DATA_BLOCK "INOUT"	// DB 80
VERSION : 0.1
  STRUCT
   I_TRO : STRUCT
    Fuse_115V_OK : BOOL ;	//115V AC OK
    Fuse_24V_OK : BOOL ;	//fuse 24V DC OK
    Overtemp_Cabinet : BOOL ;	//high temperature cabinet
    PowerBrakes_OK : BOOL ;	//Power supply brakes OK
    Power_Lift_OK : BOOL ;	//Power supply lift OK
    Power_Drum_OK : BOOL ;	//Power supply cable drum OK
    TRO_Power_Cabinet_Fan : BOOL ;	//Power supply cabinet fan OK
    TRO_Cabinet_Fan_ON : BOOL ;	//cabinet fan running
    BTN_Reset : BOOL ;	//Reset button (top cabinet)
    BTN_Preset : BOOL ;	//Preset button (3s)
    Preset_Bit_0 : BOOL ;	//Preset selection switch bit 0
    Preset_Bit_1 : BOOL ;	//Preset selection switch bit 1
    Preset_Bit_2 : BOOL ;	//Preset selection switch bit 2
    Preset_Bit_3 : BOOL ;	//Preset selection switch bit 3
    E76_6 : BOOL ;	//spare
    E76_7 : BOOL ;	//spare
    check_cableDrum_NO : BOOL ;	//check cable drum NO
    check_cableDrum_NC : BOOL ;	//check cable drum NC
    E77_2 : BOOL ;	//spar
    E77_3 : BOOL ;	//spar
    Buffer_left_Free : BOOL ;	//Buffer left occupied
    Buffer_right_Free : BOOL ;	//Buffer right occupied
    LIF_Limit_TOP : BOOL ;	//Lift limit switch top (minus)
    LIF_Limit_BOTTOM : BOOL ;	//Lift limit switch bottom (plus)
    LIF_Pos_TOP_NO : BOOL ;	//Lift limit prox. top NO
    LIF_Pos_TOP_NC : BOOL ;	//Lift limit prox. top NC
    Limit_plus : BOOL ;	//Tolley limit switch plus
    Limit_minus : BOOL ;	//Tolley limit switch minus
    FS_plus_NO : BOOL ;	//Tolley prox. switch forced slow plus NO
    FS_plus_NC : BOOL ;	//Tolley prox. switch forced slow plus NC
    FS_minus_NO : BOOL ;	//Tolley prox. switch forced slow minus NO
    FS_minus_NC : BOOL ;	//Tolley prox. switch forced slow minus NC
    SSI_Barcode_noPos : BOOL ;	//Datamatrix SSI error: no position
    SSI_Barcode_dirty : BOOL ;	//Datamatrix SSI error: dirty
    Profinet_Barcode_noPos : BOOL ;	//Datamatrix Profinet error: no position
    Profinet_Barcode_dirty : BOOL ;	//Datamatrix Profinet error: dirty
    FallProtection_Pl_1 : BOOL ;	//Trooley plus fall protection ch1
    FallProtection_Pl_2 : BOOL ;	//Trooley plus fall protection ch12
    FallProtection_Mi_1 : BOOL ;	//Trooley minus fall protection ch1
    FallProtection_Mi_2 : BOOL ;	//Trooley minus fall protection ch2
    Plus : BOOL ;	//Trolley drive plus
    Minus : BOOL ;	//Trolley drive minus
    Lift_up : BOOL ;	//Lift drive up
    Lift_down : BOOL ;	//Lift drive down
    TEL_Plus : BOOL ;	//Tellescope drive plus
    TEL_Minus : BOOL ;	//Tellescope drive minus
    E80_6 : BOOL ;	//spare
    E80_7 : BOOL ;	//spare
    spare : ARRAY  [1 .. 4 ] OF WORD ;
   END_STRUCT ;
   O_TRO : STRUCT
    A75_0 : BOOL ;	//spare
    Reset_24V : BOOL ;	//reset 24V fuses
    E75_02 : BOOL ;	//spare
    LP_Reset : BOOL ;	//lamp reset
    E75_4 : BOOL ;	//spare
    CableDrum : BOOL ;	//start cable drum
    EStop_Reset : BOOL ;	//ESTOP reset
    LP_Preset : BOOL ;	//lamp preset
    Horn : BOOL ;	//startup warning
    LP_State_0 : BOOL ;	//lamp state 0
    LP_State_1 : BOOL ;	//lamp state 1
    LP_State_2 : BOOL ;	//lamp state 2
    E76_4 : BOOL ;	//spare
    SEW_Reset : BOOL ;	//reset movi PLC
    EmergencyMode : BOOL ;	//Emergency Mode
    LIF_StartFan : BOOL ;	//startup Lift Fan
    EmergencyMode_Fwd : BOOL ;	//Emergency mode forward
    EmergencyMode_Bwd : BOOL ;	//Emergency mode backward
    A77_2 : BOOL ;	//startup Lift Fan
    A77_3 : BOOL ;	//Emergency mode forward
    A77_4 : BOOL ;	//Emergency mode backward
    A77_5 : BOOL ;	//spare
    A77_6 : BOOL ;	//spare
    A77_7 : BOOL ;	//spare
    spar_1 : BOOL ;	//spare
    spare_2 : BOOL ;	//spare
    spare_3 : BOOL ;	//spare
    spare : ARRAY  [1 .. 2 ] OF WORD ;
   END_STRUCT ;
   I_LIF : STRUCT
    E85_0 : BOOL ;	//spare
    E85_1 : BOOL ;	//spare
    E85_2 : BOOL ;	//spare
    E85_3 : BOOL ;	//spare
    error_NO : BOOL ;	//Drive telescopes error NO
    error_NC : BOOL ;	//Drive telescopes error NC
    E85_6 : BOOL ;	//spare
    E85_7 : BOOL ;	//spare
    Overload_L_NO : BOOL ;	//Overload-Monitoring left NO
    Overload_R_NO : BOOL ;	//Overload-Monitoring rigth NO
    SlapRope_L_NO : BOOL ;	//Slap-Rope-Monitoring left NO
    SlapRope_R_NO : BOOL ;	//Slap-Rope-Monitoring right NO
    E86_4 : BOOL ;	//spare
    E86_5 : BOOL ;	//spare
    TEL_Front_FirstHookOcc : BOOL ;	//hook front left occupied (1)
    TEL_Front_LastHookOcc : BOOL ;	//hook rear left occupied (2)
    TEL_Rear_FirstHookOcc : BOOL ;	//hook front right occupied (11)
    TEL_Rear_LastHookOcc : BOOL ;	//hook rear right occupied (12)
    E87_2 : BOOL ;	//spare
    E87_3 : BOOL ;	//spare
    TEL_inMidle_L : BOOL ;	//telescope left in middle position
    TEL_inMidle_R : BOOL ;	//telescope right in middle position
    E87_6 : BOOL ;	//spare
    TEL_Left_Occ_NO : BOOL ;	//telescope left occupied NO
    E88_0 : BOOL ;	//spare
    TEL_Right_Occ_NO : BOOL ;	//telescope right occupied NO
    TEL_Limit_front_NO : BOOL ;	//telescopes limit switch front NO
    TEL_Limit_front_NC : BOOL ;	//telescopes limit switch front NC
    TEL_Limit_back_NO : BOOL ;	//telescopes limit switch back NO
    TEL_Limit_back_NC : BOOL ;	//telescopes limit switch back NC
    E88_6 : BOOL ;	//spare
    E88_7 : BOOL ;	//spare
    E89_0 : BOOL ;	//spare
    E89_1 : BOOL ;	//spare
    E89_2 : BOOL ;	//spare
    E89_3 : BOOL ;	//spare
    E89_4 : BOOL ;	//spare
    E89_5 : BOOL ;	//spare
    E89_6 : BOOL ;	//spare
    E89_7 : BOOL ;	//spare
    TEL_Encoder : DINT ;	//Teleskope Encoder
   END_STRUCT ;
   O_LIF : STRUCT
    TEL_Mode1 : BOOL ;	//telescope mode_1
    TEL_Mode2 : BOOL ;	//telescope mode_2
    TEL_Start : BOOL ;	//start telescope
    TEL_Reset : BOOL ;	//reset telescope
    TEL_BCD_Bit_1 : BOOL ;	//telescope BCD Bit_1
    TEL_BCD_Bit_2 : BOOL ;	//telescope BCD Bit_2
    TEL_BCD_Bit_3 : BOOL ;	//telescope BCD Bit_3
    TEL_BCD_Bit_4 : BOOL ;	//telescope BCD Bit_4
    TEL_Light_Front_Left : BOOL ;	//lightning telescopes front left on
    TEL_Light_Front_Rigth : BOOL ;	//lightning telescopes front rigth on
    TEL_Light_Rear_Left : BOOL ;	//lightning telescopes rear Left on
    TEL_Light_Rear_Rigth : BOOL ;	//lightning telescopes rigth on
    TEL_Preset_Telescope : BOOL ;	//Preset Encoder Telescope
    A86_5 : BOOL ;	//spare
    A86_6 : BOOL ;	//spare
    A86_7 : BOOL ;	//spare
    A87_0 : BOOL ;	//spare
    A87_1 : BOOL ;	//spare
    A87_2 : BOOL ;	//spare
    A87_3 : BOOL ;	//spare
    A87_4 : BOOL ;	//spare
    A87_5 : BOOL ;	//spare
    A87_6 : BOOL ;	//spare
    A87_7 : BOOL ;	//spare
   END_STRUCT ;
  END_STRUCT ;	
BEGIN
   I_TRO.Fuse_24V_OK := TRUE;
   I_TRO.PowerBrakes_OK := TRUE;
   I_TRO.Power_Lift_OK := TRUE;
   I_TRO.Power_Drum_OK := TRUE;
   I_TRO.TRO_Power_Cabinet_Fan := TRUE;
   I_TRO.TRO_Cabinet_Fan_ON := TRUE;
   I_TRO.check_cableDrum_NO := TRUE;
   I_TRO.LIF_Pos_TOP_NO := TRUE;
   O_TRO.LP_State_0 := TRUE;
   I_LIF.error_NO := TRUE;
   I_LIF.error_NC := TRUE;
   I_LIF.TEL_Front_FirstHookOcc := TRUE;
   I_LIF.TEL_Front_LastHookOcc := TRUE;
   I_LIF.TEL_inMidle_L := TRUE;
   I_LIF.TEL_inMidle_R := TRUE;
   I_LIF.TEL_Left_Occ_NO := TRUE;
   I_LIF.TEL_Right_Occ_NO := TRUE;
   I_LIF.TEL_Limit_front_NC := TRUE;
   I_LIF.TEL_Limit_back_NC := TRUE;
   O_LIF.TEL_Mode2 := TRUE;
END_DATA_BLOCK

DATA_BLOCK "DB_ActualHookdata"	// DB 92
VERSION : 0.1
  STRUCT
   Front : STRUCT
    Hook : ARRAY  [1 .. 10 ] OF UDT 102;
   END_STRUCT ;
   Rear : STRUCT
    Hook : ARRAY  [1 .. 10 ] OF UDT 102;
   END_STRUCT ;
   ActualDB_No : INT ;
  END_STRUCT ;	
BEGIN
   Front.Hook[1].HookOver := L#6716;
   Front.Hook[1].HookUnderOffset := L#115;
   Front.Hook[1].TelPos_1.TelPos := L#3;
   Front.Hook[2].HookOver := L#5745;
   Front.Hook[2].HookUnderOffset := L#115;
   Front.Hook[2].TelPos_1.TelPos := L#3;
   Front.Hook[3].HookOver := L#4775;
   Front.Hook[3].HookUnderOffset := L#115;
   Front.Hook[3].TelPos_1.TelPos := L#3;
   Front.Hook[4].HookOver := L#3805;
   Front.Hook[4].HookUnderOffset := L#115;
   Front.Hook[4].TelPos_1.TelPos := L#3;
   Front.Hook[5].HookOver := L#2835;
   Front.Hook[5].HookUnderOffset := L#115;
   Front.Hook[5].TelPos_1.TelPos := L#3;
   Front.Hook[6].HookOver := L#1865;
   Front.Hook[6].HookUnderOffset := L#115;
   Front.Hook[6].TelPos_1.TelPos := L#3;
   Rear.Hook[1].HookOver := L#6716;
   Rear.Hook[1].HookUnderOffset := L#115;
   Rear.Hook[1].TelPos_1.TelPos := L#4;
   Rear.Hook[2].HookOver := L#5745;
   Rear.Hook[2].HookUnderOffset := L#115;
   Rear.Hook[2].TelPos_1.TelPos := L#4;
   Rear.Hook[3].HookOver := L#4775;
   Rear.Hook[3].HookUnderOffset := L#115;
   Rear.Hook[3].TelPos_1.TelPos := L#4;
   Rear.Hook[4].HookOver := L#3805;
   Rear.Hook[4].HookUnderOffset := L#115;
   Rear.Hook[4].TelPos_1.TelPos := L#4;
   Rear.Hook[5].HookOver := L#2835;
   Rear.Hook[5].HookUnderOffset := L#115;
   Rear.Hook[5].TelPos_1.TelPos := L#4;
   Rear.Hook[6].HookOver := L#1865;
   Rear.Hook[6].HookUnderOffset := L#115;
   Rear.Hook[6].TelPos_1.TelPos := L#4;
   ActualDB_No := 252;
END_DATA_BLOCK

DATA_BLOCK "Moves"	// DB 101
VERSION : 0.1
  STRUCT
   PC : UDT 7;
   Unit : ARRAY  [1 .. 50 ] OF UDT 7;
  END_STRUCT ;	
BEGIN
   PC.MsgCounter := 648;
   PC.Action := 4;
   PC.Value_01 := 5;
   PC.Value_02 := 8;
   PC.Value_03 := 100;
   PC.Value_04 := 100;
   Unit[1].Action := 4;
   Unit[1].Value_01 := 5;
   Unit[1].Value_02 := 8;
   Unit[1].Value_03 := 100;
   Unit[1].Value_04 := 100;
END_DATA_BLOCK

DATA_BLOCK "InstanzDB PNIODiag"	// DB 126
AUTHOR : ICom
FAMILY : DIAGNOSE
VERSION : 0.0
"PNIODiag"
BEGIN
END_DATA_BLOCK

DATA_BLOCK "InstanzDB STATDiag"	// DB 127
AUTHOR : ICom
FAMILY : DIAGNOSE
VERSION : 0.0
"STATDiag"
BEGIN
END_DATA_BLOCK

DATA_BLOCK "DB_Crane"	// DB 130
VERSION : 0.1
  STRUCT
   NoOfRows : INT  := 3;
   NoOfTowers : INT  := 13;
   NoOfPositions : INT  := 16;
   MoveCounts : DINT ;
   WorkingHours : DINT ;
   RemainigServiceHours : DINT ;
   CraneType : INT ;
   UnitNumber : INT ;
   Reserve9 : INT ;
   Reserve10 : INT ;
   Reserve11 : INT ;
   Reserve12 : INT ;
  END_STRUCT ;	
BEGIN
   NoOfRows := 3;
   NoOfTowers := 11;
   NoOfPositions := 16;
END_DATA_BLOCK

DATA_BLOCK "DB_Steps"	// DB 132
VERSION : 0.1
  STRUCT
   _DINT : STRUCT
    StepsStartet : DINT ;
    StepsFinished : DINT ;
    _02 : DINT ;
    _03 : DINT ;
    _04 : DINT ;
    _05 : DINT ;
    _06 : DINT ;
    _07 : DINT ;
    _08 : DINT ;
    _09 : DINT ;
    _10 : DINT ;
    _11 : DINT ;
    _12 : DINT ;
    _13 : DINT ;
    _14 : DINT ;
    _15 : DINT ;
    _16 : DINT ;
    _17 : DINT ;
    _18 : DINT ;
    _19 : DINT ;
    _20 : DINT ;
    _21 : DINT ;
    _22 : DINT ;
    _23 : DINT ;
    _24 : DINT ;
    _25 : DINT ;
    _26 : DINT ;
    _27 : DINT ;
    _28 : DINT ;
    _29 : DINT ;
    _30 : DINT ;
    _31 : DINT ;
    _32 : DINT ;
    _33 : DINT ;
    _34 : DINT ;
    _35 : DINT ;
    _36 : DINT ;
    _37 : DINT ;
    _38 : DINT ;
    _39 : DINT ;
    _40 : DINT ;
    _41 : DINT ;
    _42 : DINT ;
    _43 : DINT ;
    _44 : DINT ;
    _45 : DINT ;
    _46 : DINT ;
    _47 : DINT ;
    _48 : DINT ;
    _49 : DINT ;
    _50 : DINT ;
    _51 : DINT ;
    _52 : DINT ;
    _53 : DINT ;
    _54 : DINT ;
    _55 : DINT ;
    _56 : DINT ;
    _57 : DINT ;
    _58 : DINT ;
    _59 : DINT ;
    _60 : DINT ;
    _61 : DINT ;
    _62 : DINT ;
    _63 : DINT ;
    _64 : DINT ;
    _65 : DINT ;
    _66 : DINT ;
    _67 : DINT ;
    _68 : DINT ;
    _69 : DINT ;
    _70 : DINT ;
    _71 : DINT ;
    _72 : DINT ;
    _73 : DINT ;
    _74 : DINT ;
    _75 : DINT ;
    _76 : DINT ;
    _77 : DINT ;
    _78 : DINT ;
    _79 : DINT ;
    _80 : DINT ;
    _81 : DINT ;
    _82 : DINT ;
    _83 : DINT ;
    _84 : DINT ;
    _85 : DINT ;
    _86 : DINT ;
    _87 : DINT ;
    _88 : DINT ;
    _89 : DINT ;
    _90 : DINT ;
    _91 : DINT ;
    _92 : DINT ;
    _93 : DINT ;
    _94 : DINT ;
    _95 : DINT ;
    _96 : DINT ;
    _97 : DINT ;
    _98 : DINT ;
    _99 : DINT ;
    _100 : DINT ;
    _101 : DINT ;
    _102 : DINT ;
    _103 : DINT ;
    _104 : DINT ;
    _105 : DINT ;
    _106 : DINT ;
    _107 : DINT ;
    _108 : DINT ;
    _109 : DINT ;
    _110 : DINT ;
    _111 : DINT ;
    _112 : DINT ;
    _113 : DINT ;
    _114 : DINT ;
    _115 : DINT ;
    _116 : DINT ;
    _117 : DINT ;
    _118 : DINT ;
    _119 : DINT ;
    _120 : DINT ;
    _121 : DINT ;
    _122 : DINT ;
    _123 : DINT ;
    _124 : DINT ;
    _125 : DINT ;
    _126 : DINT ;
    _127 : DINT ;
    _128 : DINT ;
    _129 : DINT ;
    _130 : DINT ;
    _131 : DINT ;
    _132 : DINT ;
    _133 : DINT ;
    _134 : DINT ;
    _135 : DINT ;
    _136 : DINT ;
    _137 : DINT ;
    _138 : DINT ;
    _139 : DINT ;
    _140 : DINT ;
    _141 : DINT ;
    _142 : DINT ;
    _143 : DINT ;
    _144 : DINT ;
    _145 : DINT ;
    _146 : DINT ;
    _147 : DINT ;
    _148 : DINT ;
    _149 : DINT ;
    _150 : DINT ;
    _151 : DINT ;
    _152 : DINT ;
    _153 : DINT ;
    _154 : DINT ;
    _155 : DINT ;
    _156 : DINT ;
    _157 : DINT ;
    _158 : DINT ;
    _159 : DINT ;
   END_STRUCT ;
   _INT : STRUCT
    BASEPOS_Steps : INT ;
    EMPTY_Steps : INT ;
    GET_Steps : INT ;
    PUT_Steps : INT ;
    _04 : INT ;
    _05 : INT ;
    _06 : INT ;
    _07 : INT ;
    _08 : INT ;
    _09 : INT ;
    ChkHookOccCntGET : INT ;	//Check occupation sensors hook
    ChkHookOccCntPUT : INT ;
    _12 : INT ;
    _13 : INT ;
    _14 : INT ;
    _15 : INT ;
    _16 : INT ;
    _17 : INT ;
    _18 : INT ;
    _19 : INT ;
    _20 : INT ;
    _21 : INT ;
    _22 : INT ;
    _23 : INT ;
    _24 : INT ;
    _25 : INT ;
    _26 : INT ;
    _27 : INT ;
    _28 : INT ;
    _29 : INT ;
    _30 : INT ;
    _31 : INT ;
    _32 : INT ;
    _33 : INT ;
    _34 : INT ;
    _35 : INT ;
    _36 : INT ;
    _37 : INT ;
    _38 : INT ;
    _39 : INT ;
    _40 : INT ;
    _41 : INT ;
    _42 : INT ;
    _43 : INT ;
    _44 : INT ;
    _45 : INT ;
    _46 : INT ;
    _47 : INT ;
    _48 : INT ;
    _49 : INT ;
    _50 : INT ;
    _51 : INT ;
    _52 : INT ;
    _53 : INT ;
    _54 : INT ;
    _55 : INT ;
    _56 : INT ;
    _57 : INT ;
    _58 : INT ;
    _59 : INT ;
    _60 : INT ;
    _61 : INT ;
    _62 : INT ;
    _63 : INT ;
    _64 : INT ;
    _65 : INT ;
    _66 : INT ;
    _67 : INT ;
    _68 : INT ;
    _69 : INT ;
    _70 : INT ;
    _71 : INT ;
    _72 : INT ;
    _73 : INT ;
    _74 : INT ;
    _75 : INT ;
    _76 : INT ;
    _77 : INT ;
    _78 : INT ;
    _79 : INT ;
    _80 : INT ;
    _81 : INT ;
    _82 : INT ;
    _83 : INT ;
    _84 : INT ;
    _85 : INT ;
    _86 : INT ;
    _87 : INT ;
    _88 : INT ;
    _89 : INT ;
    _90 : INT ;
    _91 : INT ;
    _92 : INT ;
    _93 : INT ;
    _94 : INT ;
    _95 : INT ;
    _96 : INT ;
    _97 : INT ;
    _98 : INT ;
    _99 : INT ;
    _100 : INT ;
    _101 : INT ;
    _102 : INT ;
    _103 : INT ;
    _104 : INT ;
    _105 : INT ;
    _106 : INT ;
    _107 : INT ;
    _108 : INT ;
    _109 : INT ;
    _110 : INT ;
    _111 : INT ;
    _112 : INT ;
    _113 : INT ;
    _114 : INT ;
    _115 : INT ;
    _116 : INT ;
    _117 : INT ;
    _118 : INT ;
    _119 : INT ;
    _120 : INT ;
    _121 : INT ;
    _122 : INT ;
    _123 : INT ;
    _124 : INT ;
    _125 : INT ;
    _126 : INT ;
    _127 : INT ;
    _128 : INT ;
    _129 : INT ;
    _130 : INT ;
    _131 : INT ;
    _132 : INT ;
    _133 : INT ;
    _134 : INT ;
    _135 : INT ;
    _136 : INT ;
    _137 : INT ;
    _138 : INT ;
    _139 : INT ;
    _140 : INT ;
    _141 : INT ;
    _142 : INT ;
    _143 : INT ;
    _144 : INT ;
    _145 : INT ;
    _146 : INT ;
    _147 : INT ;
    _148 : INT ;
    _149 : INT ;
    _150 : INT ;
    _151 : INT ;
    _152 : INT ;
    _153 : INT ;
    _154 : INT ;
    _155 : INT ;
    _156 : INT ;
    _157 : INT ;
    _158 : INT ;
    _159 : INT ;
   END_STRUCT ;
   _BOOL : STRUCT
    Target_DataOK : BOOL ;
    _01 : BOOL ;
    _02 : BOOL ;
    _03 : BOOL ;
    _04 : BOOL ;
    _05 : BOOL ;
    _06 : BOOL ;
    _07 : BOOL ;
    BASEPOS_Req : BOOL ;
    EMPTY_Req : BOOL ;
    GET_Req : BOOL ;
    PUT_Req : BOOL ;
    BASEPOS_active : BOOL ;
    EMPTY_active : BOOL ;
    GET_active : BOOL ;
    PUT_active : BOOL ;
    STEPS_active : BOOL ;
    STEPS_start : BOOL ;
    GET_Finished : BOOL ;
    _19 : BOOL ;
    _20 : BOOL ;
    _21 : BOOL ;
    _22 : BOOL ;
    _23 : BOOL ;
    _24 : BOOL ;
    _25 : BOOL ;
    _26 : BOOL ;
    _27 : BOOL ;
    _28 : BOOL ;
    _29 : BOOL ;
    _30 : BOOL ;
    _31 : BOOL ;
    ChkHookOccGET : BOOL ;
    ChkHookOccGET_End : BOOL ;
    ChkHookOccGET_OK : BOOL ;
    ChkHookOccPUT : BOOL ;
    ChkHookOccPUT_End : BOOL ;
    ChkHookOccPUT_OK : BOOL ;
    ChkHookOcxGET_enable : BOOL ;
    ChkHookOcxPUT_enable : BOOL ;
    _40 : BOOL ;
    _41 : BOOL ;
    _42 : BOOL ;
    _43 : BOOL ;
    _44 : BOOL ;
    _45 : BOOL ;
    _46 : BOOL ;
    _47 : BOOL ;
    _48 : BOOL ;
    _49 : BOOL ;
    _50 : BOOL ;
    _51 : BOOL ;
    _52 : BOOL ;
    _53 : BOOL ;
    _54 : BOOL ;
    _55 : BOOL ;
    _56 : BOOL ;
    _57 : BOOL ;
    _58 : BOOL ;
    _59 : BOOL ;
    _60 : BOOL ;
    _61 : BOOL ;
    _62 : BOOL ;
    _63 : BOOL ;
    _64 : BOOL ;
    _65 : BOOL ;
    _66 : BOOL ;
    _67 : BOOL ;
    _68 : BOOL ;
    _69 : BOOL ;
    _70 : BOOL ;
    _71 : BOOL ;
    _72 : BOOL ;
    _73 : BOOL ;
    _74 : BOOL ;
    _75 : BOOL ;
    _76 : BOOL ;
    _77 : BOOL ;
    _78 : BOOL ;
    _79 : BOOL ;
    _80 : BOOL ;
    _81 : BOOL ;
    _82 : BOOL ;
    _83 : BOOL ;
    _84 : BOOL ;
    _85 : BOOL ;
    _86 : BOOL ;
    _87 : BOOL ;
    _88 : BOOL ;
    _89 : BOOL ;
    _90 : BOOL ;
    _91 : BOOL ;
    _92 : BOOL ;
    _93 : BOOL ;
    _94 : BOOL ;
    _95 : BOOL ;
    _96 : BOOL ;
    _97 : BOOL ;
    _98 : BOOL ;
    _99 : BOOL ;
    _100 : BOOL ;
    _101 : BOOL ;
    _102 : BOOL ;
    _103 : BOOL ;
    _104 : BOOL ;
    _105 : BOOL ;
    _106 : BOOL ;
    _107 : BOOL ;
    _108 : BOOL ;
    _109 : BOOL ;
    _110 : BOOL ;
    _111 : BOOL ;
    _112 : BOOL ;
    _113 : BOOL ;
    _114 : BOOL ;
    _115 : BOOL ;
    _116 : BOOL ;
    _117 : BOOL ;
    _118 : BOOL ;
    _119 : BOOL ;
    _120 : BOOL ;
    _121 : BOOL ;
    _122 : BOOL ;
    _123 : BOOL ;
    _124 : BOOL ;
    _125 : BOOL ;
    _126 : BOOL ;
    _127 : BOOL ;
    _128 : BOOL ;
    _129 : BOOL ;
    _130 : BOOL ;
    _131 : BOOL ;
    _132 : BOOL ;
    _133 : BOOL ;
    _134 : BOOL ;
    _135 : BOOL ;
    _136 : BOOL ;
    _137 : BOOL ;
    _138 : BOOL ;
    _139 : BOOL ;
    _140 : BOOL ;
    _141 : BOOL ;
    _142 : BOOL ;
    _143 : BOOL ;
    _144 : BOOL ;
    _145 : BOOL ;
    _146 : BOOL ;
    _147 : BOOL ;
    _148 : BOOL ;
    _149 : BOOL ;
    _150 : BOOL ;
    _151 : BOOL ;
    _152 : BOOL ;
    _153 : BOOL ;
    _154 : BOOL ;
    _155 : BOOL ;
    _156 : BOOL ;
    _157 : BOOL ;
    _158 : BOOL ;
    _159 : BOOL ;
   END_STRUCT ;
  END_STRUCT ;	
BEGIN
   _DINT.StepsStartet := L#46754;
   _DINT.StepsFinished := L#5503;
   _INT.GET_Steps := 50;
   _INT.ChkHookOccCntGET := 5;
   _INT.ChkHookOccCntPUT := 3;
   _BOOL.GET_active := TRUE;
   _BOOL.STEPS_active := TRUE;
   _BOOL.ChkHookOcxGET_enable := TRUE;
   _BOOL.ChkHookOcxPUT_enable := TRUE;
END_DATA_BLOCK

DATA_BLOCK "DB_CylinderTypes"	// DB 133
VERSION : 0.1
  STRUCT
   Cyl : ARRAY  [1 .. 10 ] OF UDT 110;
  END_STRUCT ;	
BEGIN
   Cyl[1].Number := 1;
   Cyl[1].DiameterMin := 410;
   Cyl[1].DiameterMax := 760;
   Cyl[2].Number := 2;
   Cyl[2].DiameterMin := 810;
   Cyl[2].DiameterMax := 910;
   Cyl[3].Number := 3;
   Cyl[3].DiameterMin := 960;
   Cyl[3].DiameterMax := 1060;
   Cyl[4].Number := 4;
   Cyl[4].DiameterMin := 1110;
   Cyl[4].DiameterMax := 1110;
   Cyl[5].Number := 5;
   Cyl[5].DiameterMin := 1160;
   Cyl[5].DiameterMax := 1210;
   Cyl[6].Number := 21;
   Cyl[6].DiameterMin := 630;
   Cyl[6].DiameterMax := 630;
END_DATA_BLOCK

DATA_BLOCK "DB_Area"	// DB 150
VERSION : 0.1
  STRUCT
   CR01_Start : DINT ;
   CR01_Stop : DINT ;
   CR01_Axis : DINT ;
   CR01_Sec : DINT ;
   CR02_Start : DINT ;
   CR02_Stop : DINT ;
   CR02_Axis : DINT ;
   CR02_Sec : DINT ;
   BR01_Start : DINT ;
   BR01_Stop : DINT ;
   BR01_Axis : DINT ;
   BR01_Sec : DINT ;
   BR02_Start : DINT ;
   BR02_Stop : DINT ;
   BR02_Axis : DINT ;
   BR02_Sec : DINT ;
   BR03_Start : DINT ;
   BR03_Stop : DINT ;
   BR03_Axis : DINT ;
   BR03_Sec : DINT ;
   BR04_Start : DINT ;
   BR04_Stop : DINT ;
   BR04_Axis : DINT ;
   BR04_Sec : DINT ;
   BR05_Start : DINT ;
   BR05_Stop : DINT ;
   BR05_Axis : DINT ;
   BR05_Sec : DINT ;
   BR06_Start : DINT ;
   BR06_Stop : DINT ;
   BR06_Axis : DINT ;
   BR06_Sec : DINT ;
   BR07_Start : DINT ;
   BR07_Stop : DINT ;
   BR07_Axis : DINT ;
   BR07_Sec : DINT ;
   BR08_Start : DINT ;
   BR08_Stop : DINT ;
   BR08_Axis : DINT ;
   BR08_Sec : DINT ;
   BR09_Start : DINT ;
   BR09_Stop : DINT ;
   BR09_Axis : DINT ;
   BR09_Sec : DINT ;
   BR10_Start : DINT ;
   BR10_Stop : DINT ;
   BR10_Axis : DINT ;
   BR10_Sec : DINT ;
   BR11_Start : DINT ;
   BR11_Stop : DINT ;
   BR11_Axis : DINT ;
   BR11_Sec : DINT ;
   BR01a_Start : DINT ;
   BR01a_Stop : DINT ;
   BR01a_Axis : DINT ;
   BR01a_Sec : DINT ;
   BR02a_Start : DINT ;
   BR02a_Stop : DINT ;
   BR02a_Axis : DINT ;
   BR02a_Sec : DINT ;
   BR03a_Start : DINT ;
   BR03a_Stop : DINT ;
   BR03a_Axis : DINT ;
   BR03a_Sec : DINT ;
   BR04a_Start : DINT ;
   BR04a_Stop : DINT ;
   BR04a_Axis : DINT ;
   BR04a_Sec : DINT ;
   BR05a_Start : DINT ;
   BR05a_Stop : DINT ;
   BR05a_Axis : DINT ;
   BR05a_Sec : DINT ;
  END_STRUCT ;	
BEGIN
   CR01_Stop := L#3800;
   CR01_Sec := L#1000;
   CR02_Start := L#320000;
   CR02_Stop := L#323800;
   CR02_Axis := L#291200;
   CR02_Sec := L#1000;
   BR01_Start := L#20000;
   BR01_Stop := L#45000;
   BR01_Axis := L#16200;
   BR01_Sec := L#1000;
   BR02_Start := L#50000;
   BR02_Stop := L#75000;
   BR02_Axis := L#46200;
   BR02_Sec := L#1000;
   BR03_Start := L#80000;
   BR03_Stop := L#105000;
   BR03_Axis := L#76200;
   BR03_Sec := L#1000;
   BR04_Start := L#110000;
   BR04_Stop := L#135000;
   BR04_Axis := L#106200;
   BR04_Sec := L#1000;
   BR05_Start := L#140000;
   BR05_Stop := L#165000;
   BR05_Axis := L#136200;
   BR05_Sec := L#1000;
   BR06_Start := L#170000;
   BR06_Stop := L#195000;
   BR06_Axis := L#166200;
   BR06_Sec := L#1000;
   BR07_Start := L#200000;
   BR07_Stop := L#225000;
   BR07_Axis := L#196200;
   BR07_Sec := L#1000;
   BR08_Start := L#230000;
   BR08_Stop := L#255000;
   BR08_Axis := L#226200;
   BR08_Sec := L#1000;
   BR09_Start := L#260000;
   BR09_Stop := L#285000;
   BR09_Axis := L#256200;
   BR09_Sec := L#1000;
   BR10_Start := L#290000;
   BR10_Stop := L#315000;
   BR10_Axis := L#286200;
   BR10_Sec := L#1000;
   BR11_Start := L#380000;
   BR11_Stop := L#384450;
   BR11_Axis := L#376200;
   BR11_Sec := L#1000;
   BR01a_Start := L#330000;
   BR01a_Stop := L#333430;
   BR01a_Axis := L#297400;
   BR01a_Sec := L#1000;
   BR02a_Start := L#340000;
   BR02a_Stop := L#343430;
   BR02a_Axis := L#307400;
   BR02a_Sec := L#1000;
   BR03a_Start := L#350000;
   BR03a_Stop := L#353430;
   BR03a_Axis := L#317400;
   BR03a_Sec := L#1000;
   BR04a_Start := L#360000;
   BR04a_Stop := L#363430;
   BR04a_Axis := L#327400;
   BR04a_Sec := L#1000;
   BR05a_Start := L#370000;
   BR05a_Stop := L#373430;
   BR05a_Axis := L#337400;
   BR05a_Sec := L#1000;
END_DATA_BLOCK

DATA_BLOCK "IDB_FB190"	// DB 190
VERSION : 0.0
"CopyHookDBs"
BEGIN
END_DATA_BLOCK

DATA_BLOCK "IDB_FB190_2"	// DB 191
VERSION : 0.0
"CopyHookDBs"
BEGIN
END_DATA_BLOCK

DATA_BLOCK "IDB1_FB192"	// DB 192
VERSION : 0.0
"READ_DBL"
BEGIN
END_DATA_BLOCK

DATA_BLOCK "IDB1_FB192_2"	// DB 193
VERSION : 0.0
"READ_DBL"
BEGIN
END_DATA_BLOCK

DATA_BLOCK "TRO_Positions"	// DB 200
VERSION : 0.1
  STRUCT
   BridgePos : STRUCT
    Bridge : ARRAY  [1 .. 11 ] OF STRUCT
     Trolley : ARRAY  [1 .. 11 ] OF DINT ;
    END_STRUCT ;
   END_STRUCT ;
  END_STRUCT ;	
BEGIN
   BridgePos.Bridge[1].Trolley[1] := L#2000;
   BridgePos.Bridge[1].Trolley[2] := L#21937;
   BridgePos.Bridge[1].Trolley[3] := L#24984;
   BridgePos.Bridge[1].Trolley[4] := L#28029;
   BridgePos.Bridge[1].Trolley[5] := L#31075;
   BridgePos.Bridge[1].Trolley[6] := L#34118;
   BridgePos.Bridge[1].Trolley[7] := L#37161;
   BridgePos.Bridge[1].Trolley[8] := L#40202;
   BridgePos.Bridge[1].Trolley[9] := L#43245;
   BridgePos.Bridge[1].Trolley[10] := L#322004;
   BridgePos.Bridge[2].Trolley[1] := L#2000;
   BridgePos.Bridge[2].Trolley[2] := L#51937;
   BridgePos.Bridge[2].Trolley[3] := L#54984;
   BridgePos.Bridge[2].Trolley[4] := L#58029;
   BridgePos.Bridge[2].Trolley[5] := L#61067;
   BridgePos.Bridge[2].Trolley[6] := L#64108;
   BridgePos.Bridge[2].Trolley[7] := L#67156;
   BridgePos.Bridge[2].Trolley[8] := L#70198;
   BridgePos.Bridge[2].Trolley[9] := L#73240;
   BridgePos.Bridge[2].Trolley[10] := L#322004;
   BridgePos.Bridge[3].Trolley[1] := L#2000;
   BridgePos.Bridge[3].Trolley[2] := L#81937;
   BridgePos.Bridge[3].Trolley[3] := L#84982;
   BridgePos.Bridge[3].Trolley[4] := L#88018;
   BridgePos.Bridge[3].Trolley[5] := L#91068;
   BridgePos.Bridge[3].Trolley[6] := L#94113;
   BridgePos.Bridge[3].Trolley[7] := L#97151;
   BridgePos.Bridge[3].Trolley[8] := L#100199;
   BridgePos.Bridge[3].Trolley[9] := L#103246;
   BridgePos.Bridge[3].Trolley[10] := L#322004;
   BridgePos.Bridge[4].Trolley[1] := L#2000;
   BridgePos.Bridge[4].Trolley[2] := L#111939;
   BridgePos.Bridge[4].Trolley[3] := L#114981;
   BridgePos.Bridge[4].Trolley[4] := L#118029;
   BridgePos.Bridge[4].Trolley[5] := L#121078;
   BridgePos.Bridge[4].Trolley[6] := L#124117;
   BridgePos.Bridge[4].Trolley[7] := L#127165;
   BridgePos.Bridge[4].Trolley[8] := L#130215;
   BridgePos.Bridge[4].Trolley[9] := L#133259;
   BridgePos.Bridge[4].Trolley[10] := L#322004;
   BridgePos.Bridge[5].Trolley[1] := L#2000;
   BridgePos.Bridge[5].Trolley[2] := L#141938;
   BridgePos.Bridge[5].Trolley[3] := L#144986;
   BridgePos.Bridge[5].Trolley[4] := L#148037;
   BridgePos.Bridge[5].Trolley[5] := L#151079;
   BridgePos.Bridge[5].Trolley[6] := L#154122;
   BridgePos.Bridge[5].Trolley[7] := L#157170;
   BridgePos.Bridge[5].Trolley[8] := L#160212;
   BridgePos.Bridge[5].Trolley[9] := L#163259;
   BridgePos.Bridge[5].Trolley[10] := L#322004;
   BridgePos.Bridge[6].Trolley[1] := L#2000;
   BridgePos.Bridge[6].Trolley[2] := L#172163;
   BridgePos.Bridge[6].Trolley[3] := L#175658;
   BridgePos.Bridge[6].Trolley[4] := L#179154;
   BridgePos.Bridge[6].Trolley[5] := L#182648;
   BridgePos.Bridge[6].Trolley[6] := L#186145;
   BridgePos.Bridge[6].Trolley[7] := L#189641;
   BridgePos.Bridge[6].Trolley[8] := L#193134;
   BridgePos.Bridge[6].Trolley[10] := L#322004;
   BridgePos.Bridge[7].Trolley[1] := L#2000;
   BridgePos.Bridge[7].Trolley[2] := L#202152;
   BridgePos.Bridge[7].Trolley[3] := L#205649;
   BridgePos.Bridge[7].Trolley[4] := L#209145;
   BridgePos.Bridge[7].Trolley[5] := L#212639;
   BridgePos.Bridge[7].Trolley[6] := L#216141;
   BridgePos.Bridge[7].Trolley[7] := L#219624;
   BridgePos.Bridge[7].Trolley[8] := L#223119;
   BridgePos.Bridge[7].Trolley[10] := L#322004;
   BridgePos.Bridge[8].Trolley[1] := L#2000;
   BridgePos.Bridge[8].Trolley[2] := L#232152;
   BridgePos.Bridge[8].Trolley[3] := L#235654;
   BridgePos.Bridge[8].Trolley[4] := L#239141;
   BridgePos.Bridge[8].Trolley[5] := L#242632;
   BridgePos.Bridge[8].Trolley[6] := L#246126;
   BridgePos.Bridge[8].Trolley[7] := L#249617;
   BridgePos.Bridge[8].Trolley[8] := L#253114;
   BridgePos.Bridge[8].Trolley[10] := L#322004;
   BridgePos.Bridge[9].Trolley[1] := L#2000;
   BridgePos.Bridge[9].Trolley[2] := L#262155;
   BridgePos.Bridge[9].Trolley[3] := L#265651;
   BridgePos.Bridge[9].Trolley[4] := L#269158;
   BridgePos.Bridge[9].Trolley[5] := L#272648;
   BridgePos.Bridge[9].Trolley[6] := L#276139;
   BridgePos.Bridge[9].Trolley[7] := L#279634;
   BridgePos.Bridge[9].Trolley[8] := L#283130;
   BridgePos.Bridge[9].Trolley[10] := L#322004;
   BridgePos.Bridge[10].Trolley[1] := L#2000;
   BridgePos.Bridge[10].Trolley[2] := L#292165;
   BridgePos.Bridge[10].Trolley[3] := L#295662;
   BridgePos.Bridge[10].Trolley[4] := L#299153;
   BridgePos.Bridge[10].Trolley[5] := L#302645;
   BridgePos.Bridge[10].Trolley[6] := L#306148;
   BridgePos.Bridge[10].Trolley[7] := L#309642;
   BridgePos.Bridge[10].Trolley[8] := L#313138;
   BridgePos.Bridge[10].Trolley[10] := L#322004;
   BridgePos.Bridge[11].Trolley[1] := L#2000;
   BridgePos.Bridge[11].Trolley[2] := L#382157;
END_DATA_BLOCK

DATA_BLOCK "BR01_TR01"	// DB 201
VERSION : 0.1
  STRUCT
   Front : STRUCT
    Hook : ARRAY  [1 .. 10 ] OF UDT 102;
   END_STRUCT ;
   Rear : STRUCT
    Hook : ARRAY  [1 .. 10 ] OF UDT 102;
   END_STRUCT ;
  END_STRUCT ;	
BEGIN
   Front.Hook[1].HookOver := L#6716;
   Front.Hook[1].HookUnderOffset := L#115;
   Front.Hook[1].TelPos_1.TelPos := L#3;
   Front.Hook[2].HookOver := L#5745;
   Front.Hook[2].HookUnderOffset := L#115;
   Front.Hook[2].TelPos_1.TelPos := L#3;
   Front.Hook[3].HookOver := L#4775;
   Front.Hook[3].HookUnderOffset := L#115;
   Front.Hook[3].TelPos_1.TelPos := L#3;
   Front.Hook[4].HookOver := L#3805;
   Front.Hook[4].HookUnderOffset := L#115;
   Front.Hook[4].TelPos_1.TelPos := L#3;
   Front.Hook[5].HookOver := L#2835;
   Front.Hook[5].HookUnderOffset := L#115;
   Front.Hook[5].TelPos_1.TelPos := L#3;
   Rear.Hook[1].HookOver := L#6716;
   Rear.Hook[1].HookUnderOffset := L#115;
   Rear.Hook[1].TelPos_1.TelPos := L#4;
   Rear.Hook[2].HookOver := L#5745;
   Rear.Hook[2].HookUnderOffset := L#115;
   Rear.Hook[2].TelPos_1.TelPos := L#4;
   Rear.Hook[3].HookOver := L#4775;
   Rear.Hook[3].HookUnderOffset := L#115;
   Rear.Hook[3].TelPos_1.TelPos := L#4;
   Rear.Hook[4].HookOver := L#3805;
   Rear.Hook[4].HookUnderOffset := L#115;
   Rear.Hook[4].TelPos_1.TelPos := L#4;
   Rear.Hook[5].HookOver := L#2835;
   Rear.Hook[5].HookUnderOffset := L#115;
   Rear.Hook[5].TelPos_1.TelPos := L#4;
END_DATA_BLOCK

DATA_BLOCK "BR01_TR02"	// DB 202
VERSION : 0.1
  STRUCT
   Front : STRUCT
    Hook : ARRAY  [1 .. 10 ] OF UDT 102;
   END_STRUCT ;
   Rear : STRUCT
    Hook : ARRAY  [1 .. 10 ] OF UDT 102;
   END_STRUCT ;
  END_STRUCT ;	
BEGIN
   Front.Hook[1].HookOver := L#6716;
   Front.Hook[1].HookUnderOffset := L#115;
   Front.Hook[1].TelPos_1.TelPos := L#3;
   Front.Hook[2].HookOver := L#5745;
   Front.Hook[2].HookUnderOffset := L#115;
   Front.Hook[2].TelPos_1.TelPos := L#3;
   Front.Hook[3].HookOver := L#4775;
   Front.Hook[3].HookUnderOffset := L#115;
   Front.Hook[3].TelPos_1.TelPos := L#3;
   Front.Hook[4].HookOver := L#3805;
   Front.Hook[4].HookUnderOffset := L#115;
   Front.Hook[4].TelPos_1.TelPos := L#3;
   Front.Hook[5].HookOver := L#2835;
   Front.Hook[5].HookUnderOffset := L#115;
   Front.Hook[5].TelPos_1.TelPos := L#3;
   Front.Hook[6].HookOver := L#1865;
   Front.Hook[6].HookUnderOffset := L#115;
   Front.Hook[6].TelPos_1.TelPos := L#3;
   Rear.Hook[1].HookOver := L#6716;
   Rear.Hook[1].HookUnderOffset := L#115;
   Rear.Hook[1].TelPos_1.TelPos := L#4;
   Rear.Hook[2].HookOver := L#5745;
   Rear.Hook[2].HookUnderOffset := L#115;
   Rear.Hook[2].TelPos_1.TelPos := L#4;
   Rear.Hook[3].HookOver := L#4775;
   Rear.Hook[3].HookUnderOffset := L#115;
   Rear.Hook[3].TelPos_1.TelPos := L#4;
   Rear.Hook[4].HookOver := L#3805;
   Rear.Hook[4].HookUnderOffset := L#115;
   Rear.Hook[4].TelPos_1.TelPos := L#4;
   Rear.Hook[5].HookOver := L#2835;
   Rear.Hook[5].HookUnderOffset := L#115;
   Rear.Hook[5].TelPos_1.TelPos := L#4;
   Rear.Hook[6].HookOver := L#1865;
   Rear.Hook[6].HookUnderOffset := L#115;
   Rear.Hook[6].TelPos_1.TelPos := L#4;
END_DATA_BLOCK

DATA_BLOCK "BR01_TR03"	// DB 203
VERSION : 0.1
  STRUCT
   Front : STRUCT
    Hook : ARRAY  [1 .. 10 ] OF UDT 102;
   END_STRUCT ;
   Rear : STRUCT
    Hook : ARRAY  [1 .. 10 ] OF UDT 102;
   END_STRUCT ;
  END_STRUCT ;	
BEGIN
   Front.Hook[1].HookOver := L#6716;
   Front.Hook[1].HookUnderOffset := L#115;
   Front.Hook[1].TelPos_1.TelPos := L#3;
   Front.Hook[2].HookOver := L#5745;
   Front.Hook[2].HookUnderOffset := L#115;
   Front.Hook[2].TelPos_1.TelPos := L#3;
   Front.Hook[3].HookOver := L#4775;
   Front.Hook[3].HookUnderOffset := L#115;
   Front.Hook[3].TelPos_1.TelPos := L#3;
   Front.Hook[4].HookOver := L#3805;
   Front.Hook[4].HookUnderOffset := L#115;
   Front.Hook[4].TelPos_1.TelPos := L#3;
   Front.Hook[5].HookOver := L#2835;
   Front.Hook[5].HookUnderOffset := L#115;
   Front.Hook[5].TelPos_1.TelPos := L#3;
   Front.Hook[6].HookOver := L#1865;
   Front.Hook[6].HookUnderOffset := L#115;
   Front.Hook[6].TelPos_1.TelPos := L#3;
   Rear.Hook[1].HookOver := L#6716;
   Rear.Hook[1].HookUnderOffset := L#115;
   Rear.Hook[1].TelPos_1.TelPos := L#4;
   Rear.Hook[2].HookOver := L#5745;
   Rear.Hook[2].HookUnderOffset := L#115;
   Rear.Hook[2].TelPos_1.TelPos := L#4;
   Rear.Hook[3].HookOver := L#4775;
   Rear.Hook[3].HookUnderOffset := L#115;
   Rear.Hook[3].TelPos_1.TelPos := L#4;
   Rear.Hook[4].HookOver := L#3805;
   Rear.Hook[4].HookUnderOffset := L#115;
   Rear.Hook[4].TelPos_1.TelPos := L#4;
   Rear.Hook[5].HookOver := L#2835;
   Rear.Hook[5].HookUnderOffset := L#115;
   Rear.Hook[5].TelPos_1.TelPos := L#4;
   Rear.Hook[6].HookOver := L#1865;
   Rear.Hook[6].HookUnderOffset := L#115;
   Rear.Hook[6].TelPos_1.TelPos := L#4;
END_DATA_BLOCK

DATA_BLOCK "BR01_TR04"	// DB 204
VERSION : 0.1
  STRUCT
   Front : STRUCT
    Hook : ARRAY  [1 .. 10 ] OF UDT 102;
   END_STRUCT ;
   Rear : STRUCT
    Hook : ARRAY  [1 .. 10 ] OF UDT 102;
   END_STRUCT ;
  END_STRUCT ;	
BEGIN
   Front.Hook[1].HookOver := L#6716;
   Front.Hook[1].HookUnderOffset := L#115;
   Front.Hook[1].TelPos_1.TelPos := L#3;
   Front.Hook[2].HookOver := L#5745;
   Front.Hook[2].HookUnderOffset := L#115;
   Front.Hook[2].TelPos_1.TelPos := L#3;
   Front.Hook[3].HookOver := L#4775;
   Front.Hook[3].HookUnderOffset := L#115;
   Front.Hook[3].TelPos_1.TelPos := L#3;
   Front.Hook[4].HookOver := L#3805;
   Front.Hook[4].HookUnderOffset := L#115;
   Front.Hook[4].TelPos_1.TelPos := L#3;
   Front.Hook[5].HookOver := L#2835;
   Front.Hook[5].HookUnderOffset := L#115;
   Front.Hook[5].TelPos_1.TelPos := L#3;
   Front.Hook[6].HookOver := L#1865;
   Front.Hook[6].HookUnderOffset := L#115;
   Front.Hook[6].TelPos_1.TelPos := L#3;
   Rear.Hook[1].HookOver := L#6716;
   Rear.Hook[1].HookUnderOffset := L#115;
   Rear.Hook[1].TelPos_1.TelPos := L#4;
   Rear.Hook[2].HookOver := L#5745;
   Rear.Hook[2].HookUnderOffset := L#115;
   Rear.Hook[2].TelPos_1.TelPos := L#4;
   Rear.Hook[3].HookOver := L#4775;
   Rear.Hook[3].HookUnderOffset := L#115;
   Rear.Hook[3].TelPos_1.TelPos := L#4;
   Rear.Hook[4].HookOver := L#3805;
   Rear.Hook[4].HookUnderOffset := L#115;
   Rear.Hook[4].TelPos_1.TelPos := L#4;
   Rear.Hook[5].HookOver := L#2835;
   Rear.Hook[5].HookUnderOffset := L#115;
   Rear.Hook[5].TelPos_1.TelPos := L#4;
   Rear.Hook[6].HookOver := L#1865;
   Rear.Hook[6].HookUnderOffset := L#115;
   Rear.Hook[6].TelPos_1.TelPos := L#4;
END_DATA_BLOCK

DATA_BLOCK "BR01_TR05"	// DB 205
VERSION : 0.1
  STRUCT
   Front : STRUCT
    Hook : ARRAY  [1 .. 10 ] OF UDT 102;
   END_STRUCT ;
   Rear : STRUCT
    Hook : ARRAY  [1 .. 10 ] OF UDT 102;
   END_STRUCT ;
  END_STRUCT ;	
BEGIN
   Front.Hook[1].HookOver := L#6716;
   Front.Hook[1].HookUnderOffset := L#115;
   Front.Hook[1].TelPos_1.TelPos := L#3;
   Front.Hook[2].HookOver := L#5745;
   Front.Hook[2].HookUnderOffset := L#115;
   Front.Hook[2].TelPos_1.TelPos := L#3;
   Front.Hook[3].HookOver := L#4775;
   Front.Hook[3].HookUnderOffset := L#115;
   Front.Hook[3].TelPos_1.TelPos := L#3;
   Front.Hook[4].HookOver := L#3805;
   Front.Hook[4].HookUnderOffset := L#115;
   Front.Hook[4].TelPos_1.TelPos := L#3;
   Front.Hook[5].HookOver := L#2835;
   Front.Hook[5].HookUnderOffset := L#115;
   Front.Hook[5].TelPos_1.TelPos := L#3;
   Front.Hook[6].HookOver := L#1865;
   Front.Hook[6].HookUnderOffset := L#115;
   Front.Hook[6].TelPos_1.TelPos := L#3;
   Rear.Hook[1].HookOver := L#6716;
   Rear.Hook[1].HookUnderOffset := L#115;
   Rear.Hook[1].TelPos_1.TelPos := L#4;
   Rear.Hook[2].HookOver := L#5745;
   Rear.Hook[2].HookUnderOffset := L#115;
   Rear.Hook[2].TelPos_1.TelPos := L#4;
   Rear.Hook[3].HookOver := L#4775;
   Rear.Hook[3].HookUnderOffset := L#115;
   Rear.Hook[3].TelPos_1.TelPos := L#4;
   Rear.Hook[4].HookOver := L#3805;
   Rear.Hook[4].HookUnderOffset := L#115;
   Rear.Hook[4].TelPos_1.TelPos := L#4;
   Rear.Hook[5].HookOver := L#2835;
   Rear.Hook[5].HookUnderOffset := L#115;
   Rear.Hook[5].TelPos_1.TelPos := L#4;
   Rear.Hook[6].HookOver := L#1865;
   Rear.Hook[6].HookUnderOffset := L#115;
   Rear.Hook[6].TelPos_1.TelPos := L#4;
END_DATA_BLOCK

DATA_BLOCK "BR01_TR06"	// DB 206
VERSION : 0.1
  STRUCT
   Front : STRUCT
    Hook : ARRAY  [1 .. 10 ] OF UDT 102;
   END_STRUCT ;
   Rear : STRUCT
    Hook : ARRAY  [1 .. 10 ] OF UDT 102;
   END_STRUCT ;
  END_STRUCT ;	
BEGIN
   Front.Hook[1].HookOver := L#6716;
   Front.Hook[1].HookUnderOffset := L#115;
   Front.Hook[1].TelPos_1.TelPos := L#3;
   Front.Hook[2].HookOver := L#5745;
   Front.Hook[2].HookUnderOffset := L#115;
   Front.Hook[2].TelPos_1.TelPos := L#3;
   Front.Hook[3].HookOver := L#4775;
   Front.Hook[3].HookUnderOffset := L#115;
   Front.Hook[3].TelPos_1.TelPos := L#3;
   Front.Hook[4].HookOver := L#3805;
   Front.Hook[4].HookUnderOffset := L#115;
   Front.Hook[4].TelPos_1.TelPos := L#3;
   Front.Hook[5].HookOver := L#2835;
   Front.Hook[5].HookUnderOffset := L#115;
   Front.Hook[5].TelPos_1.TelPos := L#3;
   Front.Hook[6].HookOver := L#1865;
   Front.Hook[6].HookUnderOffset := L#115;
   Front.Hook[6].TelPos_1.TelPos := L#3;
   Rear.Hook[1].HookOver := L#6716;
   Rear.Hook[1].HookUnderOffset := L#115;
   Rear.Hook[1].TelPos_1.TelPos := L#6;
   Rear.Hook[1].TelPos_2.TelPos := L#8;
   Rear.Hook[2].HookOver := L#6075;
   Rear.Hook[2].HookUnderOffset := L#115;
   Rear.Hook[2].TelPos_1.TelPos := L#6;
   Rear.Hook[2].TelPos_2.TelPos := L#8;
   Rear.Hook[3].HookOver := L#5435;
   Rear.Hook[3].HookUnderOffset := L#115;
   Rear.Hook[3].TelPos_1.TelPos := L#6;
   Rear.Hook[3].TelPos_2.TelPos := L#8;
   Rear.Hook[4].HookOver := L#4794;
   Rear.Hook[4].HookUnderOffset := L#115;
   Rear.Hook[4].TelPos_1.TelPos := L#6;
   Rear.Hook[4].TelPos_2.TelPos := L#8;
   Rear.Hook[5].HookOver := L#4154;
   Rear.Hook[5].HookUnderOffset := L#115;
   Rear.Hook[5].TelPos_1.TelPos := L#6;
   Rear.Hook[5].TelPos_2.TelPos := L#8;
   Rear.Hook[6].HookOver := L#3514;
   Rear.Hook[6].HookUnderOffset := L#115;
   Rear.Hook[6].TelPos_1.TelPos := L#6;
   Rear.Hook[6].TelPos_2.TelPos := L#8;
   Rear.Hook[7].HookOver := L#2873;
   Rear.Hook[7].HookUnderOffset := L#115;
   Rear.Hook[7].TelPos_1.TelPos := L#6;
   Rear.Hook[7].TelPos_2.TelPos := L#8;
   Rear.Hook[8].HookOver := L#2233;
   Rear.Hook[8].HookUnderOffset := L#115;
   Rear.Hook[8].TelPos_1.TelPos := L#6;
   Rear.Hook[8].TelPos_2.TelPos := L#8;
   Rear.Hook[9].HookOver := L#1593;
   Rear.Hook[9].HookUnderOffset := L#115;
   Rear.Hook[9].TelPos_1.TelPos := L#6;
   Rear.Hook[9].TelPos_2.TelPos := L#8;
END_DATA_BLOCK

DATA_BLOCK "BR01_TR07"	// DB 207
VERSION : 0.1
  STRUCT
   Front : STRUCT
    Hook : ARRAY  [1 .. 10 ] OF UDT 102;
   END_STRUCT ;
   Rear : STRUCT
    Hook : ARRAY  [1 .. 10 ] OF UDT 102;
   END_STRUCT ;
  END_STRUCT ;	
BEGIN
   Front.Hook[1].HookOver := L#6716;
   Front.Hook[1].HookUnderOffset := L#115;
   Front.Hook[1].TelPos_1.TelPos := L#5;
   Front.Hook[1].TelPos_2.TelPos := L#7;
   Front.Hook[2].HookOver := L#6075;
   Front.Hook[2].HookUnderOffset := L#115;
   Front.Hook[2].TelPos_1.TelPos := L#5;
   Front.Hook[2].TelPos_2.TelPos := L#7;
   Front.Hook[3].HookOver := L#5435;
   Front.Hook[3].HookUnderOffset := L#115;
   Front.Hook[3].TelPos_1.TelPos := L#5;
   Front.Hook[3].TelPos_2.TelPos := L#7;
   Front.Hook[4].HookOver := L#4794;
   Front.Hook[4].HookUnderOffset := L#115;
   Front.Hook[4].TelPos_1.TelPos := L#5;
   Front.Hook[4].TelPos_2.TelPos := L#7;
   Front.Hook[5].HookOver := L#4154;
   Front.Hook[5].HookUnderOffset := L#115;
   Front.Hook[5].TelPos_1.TelPos := L#5;
   Front.Hook[5].TelPos_2.TelPos := L#7;
   Front.Hook[6].HookOver := L#3514;
   Front.Hook[6].HookUnderOffset := L#126;
   Front.Hook[6].TelPos_1.TelPos := L#5;
   Front.Hook[6].TelPos_2.TelPos := L#7;
   Front.Hook[7].HookOver := L#2873;
   Front.Hook[7].HookUnderOffset := L#115;
   Front.Hook[7].TelPos_1.TelPos := L#5;
   Front.Hook[7].TelPos_2.TelPos := L#7;
   Front.Hook[8].HookOver := L#2233;
   Front.Hook[8].HookUnderOffset := L#115;
   Front.Hook[8].TelPos_1.TelPos := L#5;
   Front.Hook[8].TelPos_2.TelPos := L#7;
   Front.Hook[9].HookOver := L#1593;
   Front.Hook[9].HookUnderOffset := L#115;
   Front.Hook[9].TelPos_1.TelPos := L#5;
   Front.Hook[9].TelPos_2.TelPos := L#7;
   Rear.Hook[1].HookOver := L#6716;
   Rear.Hook[1].HookUnderOffset := L#115;
   Rear.Hook[1].TelPos_1.TelPos := L#6;
   Rear.Hook[1].TelPos_2.TelPos := L#8;
   Rear.Hook[2].HookOver := L#6075;
   Rear.Hook[2].HookUnderOffset := L#115;
   Rear.Hook[2].TelPos_1.TelPos := L#6;
   Rear.Hook[2].TelPos_2.TelPos := L#8;
   Rear.Hook[3].HookOver := L#5435;
   Rear.Hook[3].HookUnderOffset := L#115;
   Rear.Hook[3].TelPos_1.TelPos := L#6;
   Rear.Hook[3].TelPos_2.TelPos := L#8;
   Rear.Hook[4].HookOver := L#4794;
   Rear.Hook[4].HookUnderOffset := L#115;
   Rear.Hook[4].TelPos_1.TelPos := L#6;
   Rear.Hook[4].TelPos_2.TelPos := L#8;
   Rear.Hook[5].HookOver := L#4154;
   Rear.Hook[5].HookUnderOffset := L#115;
   Rear.Hook[5].TelPos_1.TelPos := L#6;
   Rear.Hook[5].TelPos_2.TelPos := L#8;
   Rear.Hook[6].HookOver := L#3514;
   Rear.Hook[6].HookUnderOffset := L#115;
   Rear.Hook[6].TelPos_1.TelPos := L#6;
   Rear.Hook[6].TelPos_2.TelPos := L#8;
   Rear.Hook[7].HookOver := L#2873;
   Rear.Hook[7].HookUnderOffset := L#115;
   Rear.Hook[7].TelPos_1.TelPos := L#6;
   Rear.Hook[7].TelPos_2.TelPos := L#8;
   Rear.Hook[8].HookOver := L#2233;
   Rear.Hook[8].HookUnderOffset := L#115;
   Rear.Hook[8].TelPos_1.TelPos := L#6;
   Rear.Hook[8].TelPos_2.TelPos := L#8;
   Rear.Hook[9].HookOver := L#1593;
   Rear.Hook[9].HookUnderOffset := L#115;
   Rear.Hook[9].TelPos_1.TelPos := L#6;
   Rear.Hook[9].TelPos_2.TelPos := L#8;
END_DATA_BLOCK

DATA_BLOCK "BR01_TR08"	// DB 208
VERSION : 0.1
  STRUCT
   Front : STRUCT
    Hook : ARRAY  [1 .. 10 ] OF UDT 102;
   END_STRUCT ;
   Rear : STRUCT
    Hook : ARRAY  [1 .. 10 ] OF UDT 102;
   END_STRUCT ;
  END_STRUCT ;	
BEGIN
   Front.Hook[1].HookOver := L#6716;
   Front.Hook[1].HookUnderOffset := L#115;
   Front.Hook[1].TelPos_1.TelPos := L#5;
   Front.Hook[1].TelPos_2.TelPos := L#7;
   Front.Hook[2].HookOver := L#6075;
   Front.Hook[2].HookUnderOffset := L#115;
   Front.Hook[2].TelPos_1.TelPos := L#5;
   Front.Hook[2].TelPos_2.TelPos := L#7;
   Front.Hook[3].HookOver := L#5435;
   Front.Hook[3].HookUnderOffset := L#115;
   Front.Hook[3].TelPos_1.TelPos := L#5;
   Front.Hook[3].TelPos_2.TelPos := L#7;
   Front.Hook[4].HookOver := L#4794;
   Front.Hook[4].HookUnderOffset := L#115;
   Front.Hook[4].TelPos_1.TelPos := L#5;
   Front.Hook[4].TelPos_2.TelPos := L#7;
   Front.Hook[5].HookOver := L#4154;
   Front.Hook[5].HookUnderOffset := L#115;
   Front.Hook[5].TelPos_1.TelPos := L#5;
   Front.Hook[5].TelPos_2.TelPos := L#7;
   Front.Hook[6].HookOver := L#3514;
   Front.Hook[6].HookUnderOffset := L#126;
   Front.Hook[6].TelPos_1.TelPos := L#5;
   Front.Hook[6].TelPos_2.TelPos := L#7;
   Front.Hook[7].HookOver := L#2873;
   Front.Hook[7].HookUnderOffset := L#115;
   Front.Hook[7].TelPos_1.TelPos := L#5;
   Front.Hook[7].TelPos_2.TelPos := L#7;
   Front.Hook[8].HookOver := L#2233;
   Front.Hook[8].HookUnderOffset := L#115;
   Front.Hook[8].TelPos_1.TelPos := L#5;
   Front.Hook[8].TelPos_2.TelPos := L#7;
   Front.Hook[9].HookOver := L#1593;
   Front.Hook[9].HookUnderOffset := L#115;
   Front.Hook[9].TelPos_1.TelPos := L#5;
   Front.Hook[9].TelPos_2.TelPos := L#7;
   Rear.Hook[1].HookOver := L#6716;
   Rear.Hook[1].HookUnderOffset := L#115;
   Rear.Hook[1].TelPos_1.TelPos := L#6;
   Rear.Hook[1].TelPos_2.TelPos := L#8;
   Rear.Hook[2].HookOver := L#6075;
   Rear.Hook[2].HookUnderOffset := L#115;
   Rear.Hook[2].TelPos_1.TelPos := L#6;
   Rear.Hook[2].TelPos_2.TelPos := L#8;
   Rear.Hook[3].HookOver := L#5435;
   Rear.Hook[3].HookUnderOffset := L#115;
   Rear.Hook[3].TelPos_1.TelPos := L#6;
   Rear.Hook[3].TelPos_2.TelPos := L#8;
   Rear.Hook[4].HookOver := L#4794;
   Rear.Hook[4].HookUnderOffset := L#115;
   Rear.Hook[4].TelPos_1.TelPos := L#6;
   Rear.Hook[4].TelPos_2.TelPos := L#8;
   Rear.Hook[5].HookOver := L#4154;
   Rear.Hook[5].HookUnderOffset := L#115;
   Rear.Hook[5].TelPos_1.TelPos := L#6;
   Rear.Hook[5].TelPos_2.TelPos := L#8;
   Rear.Hook[6].HookOver := L#3514;
   Rear.Hook[6].HookUnderOffset := L#115;
   Rear.Hook[6].TelPos_1.TelPos := L#6;
   Rear.Hook[6].TelPos_2.TelPos := L#8;
   Rear.Hook[7].HookOver := L#2873;
   Rear.Hook[7].HookUnderOffset := L#115;
   Rear.Hook[7].TelPos_1.TelPos := L#6;
   Rear.Hook[7].TelPos_2.TelPos := L#8;
   Rear.Hook[8].HookOver := L#2233;
   Rear.Hook[8].HookUnderOffset := L#115;
   Rear.Hook[8].TelPos_1.TelPos := L#6;
   Rear.Hook[8].TelPos_2.TelPos := L#8;
   Rear.Hook[9].HookOver := L#1593;
   Rear.Hook[9].HookUnderOffset := L#115;
   Rear.Hook[9].TelPos_1.TelPos := L#6;
   Rear.Hook[9].TelPos_2.TelPos := L#8;
END_DATA_BLOCK

DATA_BLOCK "BR01_TR09"	// DB 209
VERSION : 0.1
  STRUCT
   Front : STRUCT
    Hook : ARRAY  [1 .. 10 ] OF UDT 102;
   END_STRUCT ;
   Rear : STRUCT
    Hook : ARRAY  [1 .. 10 ] OF UDT 102;
   END_STRUCT ;
  END_STRUCT ;	
BEGIN
   Front.Hook[1].HookOver := L#6716;
   Front.Hook[1].HookUnderOffset := L#115;
   Front.Hook[1].TelPos_1.TelPos := L#5;
   Front.Hook[1].TelPos_2.TelPos := L#7;
   Front.Hook[2].HookOver := L#6075;
   Front.Hook[2].HookUnderOffset := L#115;
   Front.Hook[2].TelPos_1.TelPos := L#5;
   Front.Hook[2].TelPos_2.TelPos := L#7;
   Front.Hook[3].HookOver := L#5435;
   Front.Hook[3].HookUnderOffset := L#115;
   Front.Hook[3].TelPos_1.TelPos := L#5;
   Front.Hook[3].TelPos_2.TelPos := L#7;
   Front.Hook[4].HookOver := L#4794;
   Front.Hook[4].HookUnderOffset := L#115;
   Front.Hook[4].TelPos_1.TelPos := L#5;
   Front.Hook[4].TelPos_2.TelPos := L#7;
   Front.Hook[5].HookOver := L#4154;
   Front.Hook[5].HookUnderOffset := L#115;
   Front.Hook[5].TelPos_1.TelPos := L#5;
   Front.Hook[5].TelPos_2.TelPos := L#7;
   Front.Hook[6].HookOver := L#3514;
   Front.Hook[6].HookUnderOffset := L#126;
   Front.Hook[6].TelPos_1.TelPos := L#5;
   Front.Hook[6].TelPos_2.TelPos := L#7;
   Front.Hook[7].HookOver := L#2873;
   Front.Hook[7].HookUnderOffset := L#115;
   Front.Hook[7].TelPos_1.TelPos := L#5;
   Front.Hook[7].TelPos_2.TelPos := L#7;
   Front.Hook[8].HookOver := L#2233;
   Front.Hook[8].HookUnderOffset := L#115;
   Front.Hook[8].TelPos_1.TelPos := L#5;
   Front.Hook[8].TelPos_2.TelPos := L#7;
   Front.Hook[9].HookOver := L#1593;
   Front.Hook[9].HookUnderOffset := L#115;
   Front.Hook[9].TelPos_1.TelPos := L#5;
   Front.Hook[9].TelPos_2.TelPos := L#7;
   Rear.Hook[1].HookOver := L#6716;
   Rear.Hook[1].HookUnderOffset := L#115;
   Rear.Hook[1].TelPos_1.TelPos := L#6;
   Rear.Hook[1].TelPos_2.TelPos := L#8;
   Rear.Hook[2].HookOver := L#6075;
   Rear.Hook[2].HookUnderOffset := L#115;
   Rear.Hook[2].TelPos_1.TelPos := L#6;
   Rear.Hook[2].TelPos_2.TelPos := L#8;
   Rear.Hook[3].HookOver := L#5435;
   Rear.Hook[3].HookUnderOffset := L#115;
   Rear.Hook[3].TelPos_1.TelPos := L#6;
   Rear.Hook[3].TelPos_2.TelPos := L#8;
   Rear.Hook[4].HookOver := L#4794;
   Rear.Hook[4].HookUnderOffset := L#115;
   Rear.Hook[4].TelPos_1.TelPos := L#6;
   Rear.Hook[4].TelPos_2.TelPos := L#8;
   Rear.Hook[5].HookOver := L#4154;
   Rear.Hook[5].HookUnderOffset := L#115;
   Rear.Hook[5].TelPos_1.TelPos := L#6;
   Rear.Hook[5].TelPos_2.TelPos := L#8;
   Rear.Hook[6].HookOver := L#3514;
   Rear.Hook[6].HookUnderOffset := L#115;
   Rear.Hook[6].TelPos_1.TelPos := L#6;
   Rear.Hook[6].TelPos_2.TelPos := L#8;
   Rear.Hook[7].HookOver := L#2873;
   Rear.Hook[7].HookUnderOffset := L#115;
   Rear.Hook[7].TelPos_1.TelPos := L#6;
   Rear.Hook[7].TelPos_2.TelPos := L#8;
   Rear.Hook[8].HookOver := L#2233;
   Rear.Hook[8].HookUnderOffset := L#115;
   Rear.Hook[8].TelPos_1.TelPos := L#6;
   Rear.Hook[8].TelPos_2.TelPos := L#8;
   Rear.Hook[9].HookOver := L#1593;
   Rear.Hook[9].HookUnderOffset := L#115;
   Rear.Hook[9].TelPos_1.TelPos := L#6;
   Rear.Hook[9].TelPos_2.TelPos := L#8;
END_DATA_BLOCK

DATA_BLOCK "BR01_TR10"	// DB 210
VERSION : 0.1
  STRUCT
   Front : STRUCT
    Hook : ARRAY  [1 .. 10 ] OF UDT 102;
   END_STRUCT ;
   Rear : STRUCT
    Hook : ARRAY  [1 .. 10 ] OF UDT 102;
   END_STRUCT ;
  END_STRUCT ;	
BEGIN
   Front.Hook[1].HookOver := L#6716;
   Front.Hook[1].HookUnderOffset := L#115;
   Front.Hook[1].TelPos_1.TelPos := L#3;
   Front.Hook[2].HookOver := L#5745;
   Front.Hook[2].HookUnderOffset := L#115;
   Front.Hook[2].TelPos_1.TelPos := L#3;
   Front.Hook[3].HookOver := L#4775;
   Front.Hook[3].HookUnderOffset := L#115;
   Front.Hook[3].TelPos_1.TelPos := L#3;
   Front.Hook[4].HookOver := L#3805;
   Front.Hook[4].HookUnderOffset := L#115;
   Front.Hook[4].TelPos_1.TelPos := L#3;
   Front.Hook[5].HookOver := L#2835;
   Front.Hook[5].HookUnderOffset := L#115;
   Front.Hook[5].TelPos_1.TelPos := L#3;
   Rear.Hook[1].HookOver := L#6716;
   Rear.Hook[1].HookUnderOffset := L#115;
   Rear.Hook[1].TelPos_1.TelPos := L#4;
   Rear.Hook[2].HookOver := L#5745;
   Rear.Hook[2].HookUnderOffset := L#115;
   Rear.Hook[2].TelPos_1.TelPos := L#4;
   Rear.Hook[3].HookOver := L#4775;
   Rear.Hook[3].HookUnderOffset := L#115;
   Rear.Hook[3].TelPos_1.TelPos := L#4;
   Rear.Hook[4].HookOver := L#3805;
   Rear.Hook[4].HookUnderOffset := L#115;
   Rear.Hook[4].TelPos_1.TelPos := L#4;
   Rear.Hook[5].HookOver := L#2835;
   Rear.Hook[5].HookUnderOffset := L#115;
   Rear.Hook[5].TelPos_1.TelPos := L#4;
END_DATA_BLOCK

DATA_BLOCK "BR01_TR11"	// DB 211
VERSION : 0.1
  STRUCT
   Front : STRUCT
    Hook : ARRAY  [1 .. 10 ] OF UDT 102;
   END_STRUCT ;
   Rear : STRUCT
    Hook : ARRAY  [1 .. 10 ] OF UDT 102;
   END_STRUCT ;
  END_STRUCT ;	
BEGIN
   Front.Hook[1].HookOver := L#6716;
   Front.Hook[1].HookUnderOffset := L#115;
   Front.Hook[1].TelPos_1.TelPos := L#5;
   Front.Hook[1].TelPos_2.TelPos := L#7;
   Front.Hook[2].HookOver := L#6075;
   Front.Hook[2].HookUnderOffset := L#115;
   Front.Hook[2].TelPos_1.TelPos := L#5;
   Front.Hook[2].TelPos_2.TelPos := L#7;
   Front.Hook[3].HookOver := L#5435;
   Front.Hook[3].HookUnderOffset := L#115;
   Front.Hook[3].TelPos_1.TelPos := L#5;
   Front.Hook[3].TelPos_2.TelPos := L#7;
   Front.Hook[4].HookOver := L#4794;
   Front.Hook[4].HookUnderOffset := L#115;
   Front.Hook[4].TelPos_1.TelPos := L#5;
   Front.Hook[4].TelPos_2.TelPos := L#7;
   Front.Hook[5].HookOver := L#4154;
   Front.Hook[5].HookUnderOffset := L#115;
   Front.Hook[5].TelPos_1.TelPos := L#5;
   Front.Hook[5].TelPos_2.TelPos := L#7;
   Front.Hook[6].HookOver := L#3514;
   Front.Hook[6].HookUnderOffset := L#126;
   Front.Hook[6].TelPos_1.TelPos := L#5;
   Front.Hook[6].TelPos_2.TelPos := L#7;
   Front.Hook[7].HookOver := L#2873;
   Front.Hook[7].HookUnderOffset := L#115;
   Front.Hook[7].TelPos_1.TelPos := L#5;
   Front.Hook[7].TelPos_2.TelPos := L#7;
   Front.Hook[8].HookOver := L#2233;
   Front.Hook[8].HookUnderOffset := L#115;
   Front.Hook[8].TelPos_1.TelPos := L#5;
   Front.Hook[8].TelPos_2.TelPos := L#7;
   Front.Hook[9].HookOver := L#1593;
   Front.Hook[9].HookUnderOffset := L#115;
   Front.Hook[9].TelPos_1.TelPos := L#5;
   Front.Hook[9].TelPos_2.TelPos := L#7;
   Rear.Hook[1].HookOver := L#6716;
   Rear.Hook[1].HookUnderOffset := L#115;
   Rear.Hook[1].TelPos_1.TelPos := L#6;
   Rear.Hook[1].TelPos_2.TelPos := L#8;
   Rear.Hook[2].HookOver := L#6075;
   Rear.Hook[2].HookUnderOffset := L#115;
   Rear.Hook[2].TelPos_1.TelPos := L#6;
   Rear.Hook[2].TelPos_2.TelPos := L#8;
   Rear.Hook[3].HookOver := L#5435;
   Rear.Hook[3].HookUnderOffset := L#115;
   Rear.Hook[3].TelPos_1.TelPos := L#6;
   Rear.Hook[3].TelPos_2.TelPos := L#8;
   Rear.Hook[4].HookOver := L#4794;
   Rear.Hook[4].HookUnderOffset := L#115;
   Rear.Hook[4].TelPos_1.TelPos := L#6;
   Rear.Hook[4].TelPos_2.TelPos := L#8;
   Rear.Hook[5].HookOver := L#4154;
   Rear.Hook[5].HookUnderOffset := L#115;
   Rear.Hook[5].TelPos_1.TelPos := L#6;
   Rear.Hook[5].TelPos_2.TelPos := L#8;
   Rear.Hook[6].HookOver := L#3514;
   Rear.Hook[6].HookUnderOffset := L#115;
   Rear.Hook[6].TelPos_1.TelPos := L#6;
   Rear.Hook[6].TelPos_2.TelPos := L#8;
   Rear.Hook[7].HookOver := L#2873;
   Rear.Hook[7].HookUnderOffset := L#115;
   Rear.Hook[7].TelPos_1.TelPos := L#6;
   Rear.Hook[7].TelPos_2.TelPos := L#8;
   Rear.Hook[8].HookOver := L#2233;
   Rear.Hook[8].HookUnderOffset := L#115;
   Rear.Hook[8].TelPos_1.TelPos := L#6;
   Rear.Hook[8].TelPos_2.TelPos := L#8;
   Rear.Hook[9].HookOver := L#1593;
   Rear.Hook[9].HookUnderOffset := L#115;
   Rear.Hook[9].TelPos_1.TelPos := L#6;
   Rear.Hook[9].TelPos_2.TelPos := L#8;
END_DATA_BLOCK

DATA_BLOCK "BR02_TR01"	// DB 212
VERSION : 0.1
  STRUCT
   Front : STRUCT
    Hook : ARRAY  [1 .. 10 ] OF UDT 102;
   END_STRUCT ;
   Rear : STRUCT
    Hook : ARRAY  [1 .. 10 ] OF UDT 102;
   END_STRUCT ;
  END_STRUCT ;	
BEGIN
   Front.Hook[1].HookOver := L#6716;
   Front.Hook[1].HookUnderOffset := L#115;
   Front.Hook[1].TelPos_1.TelPos := L#3;
   Front.Hook[2].HookOver := L#5745;
   Front.Hook[2].HookUnderOffset := L#115;
   Front.Hook[2].TelPos_1.TelPos := L#3;
   Front.Hook[3].HookOver := L#4775;
   Front.Hook[3].HookUnderOffset := L#115;
   Front.Hook[3].TelPos_1.TelPos := L#3;
   Front.Hook[4].HookOver := L#3805;
   Front.Hook[4].HookUnderOffset := L#115;
   Front.Hook[4].TelPos_1.TelPos := L#3;
   Front.Hook[5].HookOver := L#2835;
   Front.Hook[5].HookUnderOffset := L#115;
   Front.Hook[5].TelPos_1.TelPos := L#3;
   Rear.Hook[1].HookOver := L#6716;
   Rear.Hook[1].HookUnderOffset := L#115;
   Rear.Hook[1].TelPos_1.TelPos := L#4;
   Rear.Hook[2].HookOver := L#5745;
   Rear.Hook[2].HookUnderOffset := L#115;
   Rear.Hook[2].TelPos_1.TelPos := L#4;
   Rear.Hook[3].HookOver := L#4775;
   Rear.Hook[3].HookUnderOffset := L#115;
   Rear.Hook[3].TelPos_1.TelPos := L#4;
   Rear.Hook[4].HookOver := L#3805;
   Rear.Hook[4].HookUnderOffset := L#115;
   Rear.Hook[4].TelPos_1.TelPos := L#4;
   Rear.Hook[5].HookOver := L#2835;
   Rear.Hook[5].HookUnderOffset := L#115;
   Rear.Hook[5].TelPos_1.TelPos := L#4;
END_DATA_BLOCK

DATA_BLOCK "BR02_TR02"	// DB 213
VERSION : 0.1
  STRUCT
   Front : STRUCT
    Hook : ARRAY  [1 .. 10 ] OF UDT 102;
   END_STRUCT ;
   Rear : STRUCT
    Hook : ARRAY  [1 .. 10 ] OF UDT 102;
   END_STRUCT ;
  END_STRUCT ;	
BEGIN
   Front.Hook[1].HookOver := L#6716;
   Front.Hook[1].HookUnderOffset := L#115;
   Front.Hook[1].TelPos_1.TelPos := L#3;
   Front.Hook[2].HookOver := L#5745;
   Front.Hook[2].HookUnderOffset := L#115;
   Front.Hook[2].TelPos_1.TelPos := L#3;
   Front.Hook[3].HookOver := L#4775;
   Front.Hook[3].HookUnderOffset := L#115;
   Front.Hook[3].TelPos_1.TelPos := L#3;
   Front.Hook[4].HookOver := L#3805;
   Front.Hook[4].HookUnderOffset := L#115;
   Front.Hook[4].TelPos_1.TelPos := L#3;
   Front.Hook[5].HookOver := L#2835;
   Front.Hook[5].HookUnderOffset := L#115;
   Front.Hook[5].TelPos_1.TelPos := L#3;
   Front.Hook[6].HookOver := L#1865;
   Front.Hook[6].HookUnderOffset := L#115;
   Front.Hook[6].TelPos_1.TelPos := L#3;
   Rear.Hook[1].HookOver := L#6716;
   Rear.Hook[1].HookUnderOffset := L#115;
   Rear.Hook[1].TelPos_1.TelPos := L#4;
   Rear.Hook[2].HookOver := L#5745;
   Rear.Hook[2].HookUnderOffset := L#115;
   Rear.Hook[2].TelPos_1.TelPos := L#4;
   Rear.Hook[3].HookOver := L#4775;
   Rear.Hook[3].HookUnderOffset := L#115;
   Rear.Hook[3].TelPos_1.TelPos := L#4;
   Rear.Hook[4].HookOver := L#3805;
   Rear.Hook[4].HookUnderOffset := L#115;
   Rear.Hook[4].TelPos_1.TelPos := L#4;
   Rear.Hook[5].HookOver := L#2835;
   Rear.Hook[5].HookUnderOffset := L#115;
   Rear.Hook[5].TelPos_1.TelPos := L#4;
   Rear.Hook[6].HookOver := L#1865;
   Rear.Hook[6].HookUnderOffset := L#115;
   Rear.Hook[6].TelPos_1.TelPos := L#4;
END_DATA_BLOCK

DATA_BLOCK "BR02_TR03"	// DB 214
VERSION : 0.1
  STRUCT
   Front : STRUCT
    Hook : ARRAY  [1 .. 10 ] OF UDT 102;
   END_STRUCT ;
   Rear : STRUCT
    Hook : ARRAY  [1 .. 10 ] OF UDT 102;
   END_STRUCT ;
  END_STRUCT ;	
BEGIN
   Front.Hook[1].HookOver := L#6716;
   Front.Hook[1].HookUnderOffset := L#115;
   Front.Hook[1].TelPos_1.TelPos := L#3;
   Front.Hook[2].HookOver := L#5745;
   Front.Hook[2].HookUnderOffset := L#115;
   Front.Hook[2].TelPos_1.TelPos := L#3;
   Front.Hook[3].HookOver := L#4775;
   Front.Hook[3].HookUnderOffset := L#115;
   Front.Hook[3].TelPos_1.TelPos := L#3;
   Front.Hook[4].HookOver := L#3805;
   Front.Hook[4].HookUnderOffset := L#115;
   Front.Hook[4].TelPos_1.TelPos := L#3;
   Front.Hook[5].HookOver := L#2835;
   Front.Hook[5].HookUnderOffset := L#115;
   Front.Hook[5].TelPos_1.TelPos := L#3;
   Front.Hook[6].HookOver := L#1865;
   Front.Hook[6].HookUnderOffset := L#115;
   Front.Hook[6].TelPos_1.TelPos := L#3;
   Rear.Hook[1].HookOver := L#6716;
   Rear.Hook[1].HookUnderOffset := L#115;
   Rear.Hook[1].TelPos_1.TelPos := L#4;
   Rear.Hook[2].HookOver := L#5745;
   Rear.Hook[2].HookUnderOffset := L#115;
   Rear.Hook[2].TelPos_1.TelPos := L#4;
   Rear.Hook[3].HookOver := L#4775;
   Rear.Hook[3].HookUnderOffset := L#115;
   Rear.Hook[3].TelPos_1.TelPos := L#4;
   Rear.Hook[4].HookOver := L#3805;
   Rear.Hook[4].HookUnderOffset := L#115;
   Rear.Hook[4].TelPos_1.TelPos := L#4;
   Rear.Hook[5].HookOver := L#2835;
   Rear.Hook[5].HookUnderOffset := L#115;
   Rear.Hook[5].TelPos_1.TelPos := L#4;
   Rear.Hook[6].HookOver := L#1865;
   Rear.Hook[6].HookUnderOffset := L#115;
   Rear.Hook[6].TelPos_1.TelPos := L#4;
END_DATA_BLOCK

DATA_BLOCK "BR02_TR04"	// DB 215
VERSION : 0.1
  STRUCT
   Front : STRUCT
    Hook : ARRAY  [1 .. 10 ] OF UDT 102;
   END_STRUCT ;
   Rear : STRUCT
    Hook : ARRAY  [1 .. 10 ] OF UDT 102;
   END_STRUCT ;
  END_STRUCT ;	
BEGIN
   Front.Hook[1].HookOver := L#6716;
   Front.Hook[1].HookUnderOffset := L#115;
   Front.Hook[1].TelPos_1.TelPos := L#3;
   Front.Hook[2].HookOver := L#5745;
   Front.Hook[2].HookUnderOffset := L#115;
   Front.Hook[2].TelPos_1.TelPos := L#3;
   Front.Hook[3].HookOver := L#4775;
   Front.Hook[3].HookUnderOffset := L#115;
   Front.Hook[3].TelPos_1.TelPos := L#3;
   Front.Hook[4].HookOver := L#3805;
   Front.Hook[4].HookUnderOffset := L#115;
   Front.Hook[4].TelPos_1.TelPos := L#3;
   Front.Hook[5].HookOver := L#2835;
   Front.Hook[5].HookUnderOffset := L#115;
   Front.Hook[5].TelPos_1.TelPos := L#3;
   Front.Hook[6].HookOver := L#1865;
   Front.Hook[6].HookUnderOffset := L#115;
   Front.Hook[6].TelPos_1.TelPos := L#3;
   Rear.Hook[1].HookOver := L#6716;
   Rear.Hook[1].HookUnderOffset := L#115;
   Rear.Hook[1].TelPos_1.TelPos := L#4;
   Rear.Hook[2].HookOver := L#5745;
   Rear.Hook[2].HookUnderOffset := L#115;
   Rear.Hook[2].TelPos_1.TelPos := L#4;
   Rear.Hook[3].HookOver := L#4775;
   Rear.Hook[3].HookUnderOffset := L#115;
   Rear.Hook[3].TelPos_1.TelPos := L#4;
   Rear.Hook[4].HookOver := L#3805;
   Rear.Hook[4].HookUnderOffset := L#115;
   Rear.Hook[4].TelPos_1.TelPos := L#4;
   Rear.Hook[5].HookOver := L#2835;
   Rear.Hook[5].HookUnderOffset := L#115;
   Rear.Hook[5].TelPos_1.TelPos := L#4;
   Rear.Hook[6].HookOver := L#1865;
   Rear.Hook[6].HookUnderOffset := L#115;
   Rear.Hook[6].TelPos_1.TelPos := L#4;
END_DATA_BLOCK

DATA_BLOCK "BR02_TR05"	// DB 216
VERSION : 0.1
  STRUCT
   Front : STRUCT
    Hook : ARRAY  [1 .. 10 ] OF UDT 102;
   END_STRUCT ;
   Rear : STRUCT
    Hook : ARRAY  [1 .. 10 ] OF UDT 102;
   END_STRUCT ;
  END_STRUCT ;	
BEGIN
   Front.Hook[1].HookOver := L#6716;
   Front.Hook[1].HookUnderOffset := L#115;
   Front.Hook[1].TelPos_1.TelPos := L#3;
   Front.Hook[2].HookOver := L#5745;
   Front.Hook[2].HookUnderOffset := L#115;
   Front.Hook[2].TelPos_1.TelPos := L#3;
   Front.Hook[3].HookOver := L#4775;
   Front.Hook[3].HookUnderOffset := L#115;
   Front.Hook[3].TelPos_1.TelPos := L#3;
   Front.Hook[4].HookOver := L#3805;
   Front.Hook[4].HookUnderOffset := L#115;
   Front.Hook[4].TelPos_1.TelPos := L#3;
   Front.Hook[5].HookOver := L#2835;
   Front.Hook[5].HookUnderOffset := L#115;
   Front.Hook[5].TelPos_1.TelPos := L#3;
   Front.Hook[6].HookOver := L#1865;
   Front.Hook[6].HookUnderOffset := L#115;
   Front.Hook[6].TelPos_1.TelPos := L#3;
   Rear.Hook[1].HookOver := L#6716;
   Rear.Hook[1].HookUnderOffset := L#115;
   Rear.Hook[1].TelPos_1.TelPos := L#4;
   Rear.Hook[2].HookOver := L#5745;
   Rear.Hook[2].HookUnderOffset := L#115;
   Rear.Hook[2].TelPos_1.TelPos := L#4;
   Rear.Hook[3].HookOver := L#4775;
   Rear.Hook[3].HookUnderOffset := L#115;
   Rear.Hook[3].TelPos_1.TelPos := L#4;
   Rear.Hook[4].HookOver := L#3805;
   Rear.Hook[4].HookUnderOffset := L#115;
   Rear.Hook[4].TelPos_1.TelPos := L#4;
   Rear.Hook[5].HookOver := L#2835;
   Rear.Hook[5].HookUnderOffset := L#115;
   Rear.Hook[5].TelPos_1.TelPos := L#4;
   Rear.Hook[6].HookOver := L#1865;
   Rear.Hook[6].HookUnderOffset := L#115;
   Rear.Hook[6].TelPos_1.TelPos := L#4;
END_DATA_BLOCK

DATA_BLOCK "BR02_TR06"	// DB 217
VERSION : 0.1
  STRUCT
   Front : STRUCT
    Hook : ARRAY  [1 .. 10 ] OF UDT 102;
   END_STRUCT ;
   Rear : STRUCT
    Hook : ARRAY  [1 .. 10 ] OF UDT 102;
   END_STRUCT ;
  END_STRUCT ;	
BEGIN
   Front.Hook[1].HookOver := L#6716;
   Front.Hook[1].HookUnderOffset := L#115;
   Front.Hook[1].TelPos_1.TelPos := L#3;
   Front.Hook[2].HookOver := L#5745;
   Front.Hook[2].HookUnderOffset := L#115;
   Front.Hook[2].TelPos_1.TelPos := L#3;
   Front.Hook[3].HookOver := L#4775;
   Front.Hook[3].HookUnderOffset := L#115;
   Front.Hook[3].TelPos_1.TelPos := L#3;
   Front.Hook[4].HookOver := L#3805;
   Front.Hook[4].HookUnderOffset := L#115;
   Front.Hook[4].TelPos_1.TelPos := L#3;
   Front.Hook[5].HookOver := L#2835;
   Front.Hook[5].HookUnderOffset := L#115;
   Front.Hook[5].TelPos_1.TelPos := L#3;
   Front.Hook[6].HookOver := L#1865;
   Front.Hook[6].HookUnderOffset := L#115;
   Front.Hook[6].TelPos_1.TelPos := L#3;
   Rear.Hook[1].HookOver := L#6716;
   Rear.Hook[1].HookUnderOffset := L#115;
   Rear.Hook[1].TelPos_1.TelPos := L#4;
   Rear.Hook[2].HookOver := L#5745;
   Rear.Hook[2].HookUnderOffset := L#115;
   Rear.Hook[2].TelPos_1.TelPos := L#4;
   Rear.Hook[3].HookOver := L#4775;
   Rear.Hook[3].HookUnderOffset := L#115;
   Rear.Hook[3].TelPos_1.TelPos := L#4;
   Rear.Hook[4].HookOver := L#3805;
   Rear.Hook[4].HookUnderOffset := L#115;
   Rear.Hook[4].TelPos_1.TelPos := L#4;
   Rear.Hook[5].HookOver := L#2835;
   Rear.Hook[5].HookUnderOffset := L#115;
   Rear.Hook[5].TelPos_1.TelPos := L#4;
   Rear.Hook[6].HookOver := L#1865;
   Rear.Hook[6].HookUnderOffset := L#115;
   Rear.Hook[6].TelPos_1.TelPos := L#4;
END_DATA_BLOCK

DATA_BLOCK "BR02_TR07"	// DB 218
VERSION : 0.1
  STRUCT
   Front : STRUCT
    Hook : ARRAY  [1 .. 10 ] OF UDT 102;
   END_STRUCT ;
   Rear : STRUCT
    Hook : ARRAY  [1 .. 10 ] OF UDT 102;
   END_STRUCT ;
  END_STRUCT ;	
BEGIN
   Front.Hook[1].HookOver := L#6716;
   Front.Hook[1].HookUnderOffset := L#115;
   Front.Hook[1].TelPos_1.TelPos := L#3;
   Front.Hook[2].HookOver := L#5745;
   Front.Hook[2].HookUnderOffset := L#115;
   Front.Hook[2].TelPos_1.TelPos := L#3;
   Front.Hook[3].HookOver := L#4775;
   Front.Hook[3].HookUnderOffset := L#115;
   Front.Hook[3].TelPos_1.TelPos := L#3;
   Front.Hook[4].HookOver := L#3805;
   Front.Hook[4].HookUnderOffset := L#115;
   Front.Hook[4].TelPos_1.TelPos := L#3;
   Front.Hook[5].HookOver := L#2835;
   Front.Hook[5].HookUnderOffset := L#115;
   Front.Hook[5].TelPos_1.TelPos := L#3;
   Front.Hook[6].HookOver := L#1865;
   Front.Hook[6].HookUnderOffset := L#115;
   Front.Hook[6].TelPos_1.TelPos := L#3;
   Rear.Hook[1].HookOver := L#6716;
   Rear.Hook[1].HookUnderOffset := L#115;
   Rear.Hook[1].TelPos_1.TelPos := L#4;
   Rear.Hook[2].HookOver := L#5745;
   Rear.Hook[2].HookUnderOffset := L#115;
   Rear.Hook[2].TelPos_1.TelPos := L#4;
   Rear.Hook[3].HookOver := L#4775;
   Rear.Hook[3].HookUnderOffset := L#115;
   Rear.Hook[3].TelPos_1.TelPos := L#4;
   Rear.Hook[4].HookOver := L#3805;
   Rear.Hook[4].HookUnderOffset := L#115;
   Rear.Hook[4].TelPos_1.TelPos := L#4;
   Rear.Hook[5].HookOver := L#2835;
   Rear.Hook[5].HookUnderOffset := L#115;
   Rear.Hook[5].TelPos_1.TelPos := L#4;
   Rear.Hook[6].HookOver := L#1865;
   Rear.Hook[6].HookUnderOffset := L#115;
   Rear.Hook[6].TelPos_1.TelPos := L#4;
END_DATA_BLOCK

DATA_BLOCK "BR02_TR08"	// DB 219
VERSION : 0.1
  STRUCT
   Front : STRUCT
    Hook : ARRAY  [1 .. 10 ] OF UDT 102;
   END_STRUCT ;
   Rear : STRUCT
    Hook : ARRAY  [1 .. 10 ] OF UDT 102;
   END_STRUCT ;
  END_STRUCT ;	
BEGIN
   Front.Hook[1].HookOver := L#6716;
   Front.Hook[1].HookUnderOffset := L#115;
   Front.Hook[1].TelPos_1.TelPos := L#3;
   Front.Hook[2].HookOver := L#5745;
   Front.Hook[2].HookUnderOffset := L#115;
   Front.Hook[2].TelPos_1.TelPos := L#3;
   Front.Hook[3].HookOver := L#4775;
   Front.Hook[3].HookUnderOffset := L#115;
   Front.Hook[3].TelPos_1.TelPos := L#3;
   Front.Hook[4].HookOver := L#3805;
   Front.Hook[4].HookUnderOffset := L#115;
   Front.Hook[4].TelPos_1.TelPos := L#3;
   Front.Hook[5].HookOver := L#2835;
   Front.Hook[5].HookUnderOffset := L#115;
   Front.Hook[5].TelPos_1.TelPos := L#3;
   Front.Hook[6].HookOver := L#1865;
   Front.Hook[6].HookUnderOffset := L#115;
   Front.Hook[6].TelPos_1.TelPos := L#3;
   Rear.Hook[1].HookOver := L#6716;
   Rear.Hook[1].HookUnderOffset := L#115;
   Rear.Hook[1].TelPos_1.TelPos := L#4;
   Rear.Hook[2].HookOver := L#5745;
   Rear.Hook[2].HookUnderOffset := L#115;
   Rear.Hook[2].TelPos_1.TelPos := L#4;
   Rear.Hook[3].HookOver := L#4775;
   Rear.Hook[3].HookUnderOffset := L#115;
   Rear.Hook[3].TelPos_1.TelPos := L#4;
   Rear.Hook[4].HookOver := L#3805;
   Rear.Hook[4].HookUnderOffset := L#115;
   Rear.Hook[4].TelPos_1.TelPos := L#4;
   Rear.Hook[5].HookOver := L#2835;
   Rear.Hook[5].HookUnderOffset := L#115;
   Rear.Hook[5].TelPos_1.TelPos := L#4;
   Rear.Hook[6].HookOver := L#1865;
   Rear.Hook[6].HookUnderOffset := L#115;
   Rear.Hook[6].TelPos_1.TelPos := L#4;
END_DATA_BLOCK

DATA_BLOCK "BR02_TR09"	// DB 220
VERSION : 0.1
  STRUCT
   Front : STRUCT
    Hook : ARRAY  [1 .. 10 ] OF UDT 102;
   END_STRUCT ;
   Rear : STRUCT
    Hook : ARRAY  [1 .. 10 ] OF UDT 102;
   END_STRUCT ;
  END_STRUCT ;	
BEGIN
   Front.Hook[1].HookOver := L#6716;
   Front.Hook[1].HookUnderOffset := L#115;
   Front.Hook[1].TelPos_1.TelPos := L#3;
   Front.Hook[2].HookOver := L#5745;
   Front.Hook[2].HookUnderOffset := L#115;
   Front.Hook[2].TelPos_1.TelPos := L#3;
   Front.Hook[3].HookOver := L#4775;
   Front.Hook[3].HookUnderOffset := L#115;
   Front.Hook[3].TelPos_1.TelPos := L#3;
   Front.Hook[4].HookOver := L#3805;
   Front.Hook[4].HookUnderOffset := L#115;
   Front.Hook[4].TelPos_1.TelPos := L#3;
   Front.Hook[5].HookOver := L#2835;
   Front.Hook[5].HookUnderOffset := L#115;
   Front.Hook[5].TelPos_1.TelPos := L#3;
   Front.Hook[6].HookOver := L#1865;
   Front.Hook[6].HookUnderOffset := L#115;
   Front.Hook[6].TelPos_1.TelPos := L#3;
   Rear.Hook[1].HookOver := L#6716;
   Rear.Hook[1].HookUnderOffset := L#115;
   Rear.Hook[1].TelPos_1.TelPos := L#4;
   Rear.Hook[2].HookOver := L#5745;
   Rear.Hook[2].HookUnderOffset := L#115;
   Rear.Hook[2].TelPos_1.TelPos := L#4;
   Rear.Hook[3].HookOver := L#4775;
   Rear.Hook[3].HookUnderOffset := L#115;
   Rear.Hook[3].TelPos_1.TelPos := L#4;
   Rear.Hook[4].HookOver := L#3805;
   Rear.Hook[4].HookUnderOffset := L#115;
   Rear.Hook[4].TelPos_1.TelPos := L#4;
   Rear.Hook[5].HookOver := L#2835;
   Rear.Hook[5].HookUnderOffset := L#115;
   Rear.Hook[5].TelPos_1.TelPos := L#4;
   Rear.Hook[6].HookOver := L#1865;
   Rear.Hook[6].HookUnderOffset := L#115;
   Rear.Hook[6].TelPos_1.TelPos := L#4;
END_DATA_BLOCK

DATA_BLOCK "BR02_TR10"	// DB 221
VERSION : 0.1
  STRUCT
   Front : STRUCT
    Hook : ARRAY  [1 .. 10 ] OF UDT 102;
   END_STRUCT ;
   Rear : STRUCT
    Hook : ARRAY  [1 .. 10 ] OF UDT 102;
   END_STRUCT ;
  END_STRUCT ;	
BEGIN
   Front.Hook[1].HookOver := L#6716;
   Front.Hook[1].HookUnderOffset := L#115;
   Front.Hook[1].TelPos_1.TelPos := L#3;
   Front.Hook[2].HookOver := L#5745;
   Front.Hook[2].HookUnderOffset := L#115;
   Front.Hook[2].TelPos_1.TelPos := L#3;
   Front.Hook[3].HookOver := L#4775;
   Front.Hook[3].HookUnderOffset := L#115;
   Front.Hook[3].TelPos_1.TelPos := L#3;
   Front.Hook[4].HookOver := L#3805;
   Front.Hook[4].HookUnderOffset := L#115;
   Front.Hook[4].TelPos_1.TelPos := L#3;
   Front.Hook[5].HookOver := L#2835;
   Front.Hook[5].HookUnderOffset := L#115;
   Front.Hook[5].TelPos_1.TelPos := L#3;
   Rear.Hook[1].HookOver := L#6716;
   Rear.Hook[1].HookUnderOffset := L#115;
   Rear.Hook[1].TelPos_1.TelPos := L#4;
   Rear.Hook[2].HookOver := L#5745;
   Rear.Hook[2].HookUnderOffset := L#115;
   Rear.Hook[2].TelPos_1.TelPos := L#4;
   Rear.Hook[3].HookOver := L#4775;
   Rear.Hook[3].HookUnderOffset := L#115;
   Rear.Hook[3].TelPos_1.TelPos := L#4;
   Rear.Hook[4].HookOver := L#3805;
   Rear.Hook[4].HookUnderOffset := L#115;
   Rear.Hook[4].TelPos_1.TelPos := L#4;
   Rear.Hook[5].HookOver := L#2835;
   Rear.Hook[5].HookUnderOffset := L#115;
   Rear.Hook[5].TelPos_1.TelPos := L#4;
END_DATA_BLOCK

DATA_BLOCK "BR02_TR11"	// DB 222
VERSION : 0.1
  STRUCT
   Front : STRUCT
    Hook : ARRAY  [1 .. 10 ] OF UDT 102;
   END_STRUCT ;
   Rear : STRUCT
    Hook : ARRAY  [1 .. 10 ] OF UDT 102;
   END_STRUCT ;
  END_STRUCT ;	
BEGIN
   Front.Hook[1].HookOver := L#6716;
   Front.Hook[1].HookUnderOffset := L#115;
   Front.Hook[1].TelPos_1.TelPos := L#3;
   Front.Hook[2].HookOver := L#5745;
   Front.Hook[2].HookUnderOffset := L#115;
   Front.Hook[2].TelPos_1.TelPos := L#3;
   Front.Hook[3].HookOver := L#4775;
   Front.Hook[3].HookUnderOffset := L#115;
   Front.Hook[3].TelPos_1.TelPos := L#3;
   Front.Hook[4].HookOver := L#3805;
   Front.Hook[4].HookUnderOffset := L#115;
   Front.Hook[4].TelPos_1.TelPos := L#3;
   Front.Hook[5].HookOver := L#2835;
   Front.Hook[5].HookUnderOffset := L#115;
   Front.Hook[5].TelPos_1.TelPos := L#3;
   Front.Hook[6].HookOver := L#1865;
   Front.Hook[6].HookUnderOffset := L#115;
   Front.Hook[6].TelPos_1.TelPos := L#3;
   Rear.Hook[1].HookOver := L#6716;
   Rear.Hook[1].HookUnderOffset := L#115;
   Rear.Hook[1].TelPos_1.TelPos := L#4;
   Rear.Hook[2].HookOver := L#5745;
   Rear.Hook[2].HookUnderOffset := L#115;
   Rear.Hook[2].TelPos_1.TelPos := L#4;
   Rear.Hook[3].HookOver := L#4775;
   Rear.Hook[3].HookUnderOffset := L#115;
   Rear.Hook[3].TelPos_1.TelPos := L#4;
   Rear.Hook[4].HookOver := L#3805;
   Rear.Hook[4].HookUnderOffset := L#115;
   Rear.Hook[4].TelPos_1.TelPos := L#4;
   Rear.Hook[5].HookOver := L#2835;
   Rear.Hook[5].HookUnderOffset := L#115;
   Rear.Hook[5].TelPos_1.TelPos := L#4;
   Rear.Hook[6].HookOver := L#1865;
   Rear.Hook[6].HookUnderOffset := L#115;
   Rear.Hook[6].TelPos_1.TelPos := L#4;
END_DATA_BLOCK

DATA_BLOCK "BR03_TR01"	// DB 223
VERSION : 0.1
  STRUCT
   Front : STRUCT
    Hook : ARRAY  [1 .. 10 ] OF UDT 102;
   END_STRUCT ;
   Rear : STRUCT
    Hook : ARRAY  [1 .. 10 ] OF UDT 102;
   END_STRUCT ;
  END_STRUCT ;	
BEGIN
   Front.Hook[1].HookOver := L#6716;
   Front.Hook[1].HookUnderOffset := L#115;
   Front.Hook[1].TelPos_1.TelPos := L#3;
   Front.Hook[2].HookOver := L#5745;
   Front.Hook[2].HookUnderOffset := L#115;
   Front.Hook[2].TelPos_1.TelPos := L#3;
   Front.Hook[3].HookOver := L#4775;
   Front.Hook[3].HookUnderOffset := L#115;
   Front.Hook[3].TelPos_1.TelPos := L#3;
   Front.Hook[4].HookOver := L#3805;
   Front.Hook[4].HookUnderOffset := L#115;
   Front.Hook[4].TelPos_1.TelPos := L#3;
   Front.Hook[5].HookOver := L#2835;
   Front.Hook[5].HookUnderOffset := L#115;
   Front.Hook[5].TelPos_1.TelPos := L#3;
   Rear.Hook[1].HookOver := L#6716;
   Rear.Hook[1].HookUnderOffset := L#115;
   Rear.Hook[1].TelPos_1.TelPos := L#4;
   Rear.Hook[2].HookOver := L#5745;
   Rear.Hook[2].HookUnderOffset := L#115;
   Rear.Hook[2].TelPos_1.TelPos := L#4;
   Rear.Hook[3].HookOver := L#4775;
   Rear.Hook[3].HookUnderOffset := L#115;
   Rear.Hook[3].TelPos_1.TelPos := L#4;
   Rear.Hook[4].HookOver := L#3805;
   Rear.Hook[4].HookUnderOffset := L#115;
   Rear.Hook[4].TelPos_1.TelPos := L#4;
   Rear.Hook[5].HookOver := L#2835;
   Rear.Hook[5].HookUnderOffset := L#115;
   Rear.Hook[5].TelPos_1.TelPos := L#4;
END_DATA_BLOCK

DATA_BLOCK "BR03_TR02"	// DB 224
VERSION : 0.1
  STRUCT
   Front : STRUCT
    Hook : ARRAY  [1 .. 10 ] OF UDT 102;
   END_STRUCT ;
   Rear : STRUCT
    Hook : ARRAY  [1 .. 10 ] OF UDT 102;
   END_STRUCT ;
  END_STRUCT ;	
BEGIN
   Front.Hook[1].HookOver := L#6716;
   Front.Hook[1].HookUnderOffset := L#115;
   Front.Hook[1].TelPos_1.TelPos := L#3;
   Front.Hook[2].HookOver := L#5745;
   Front.Hook[2].HookUnderOffset := L#115;
   Front.Hook[2].TelPos_1.TelPos := L#3;
   Front.Hook[3].HookOver := L#4775;
   Front.Hook[3].HookUnderOffset := L#115;
   Front.Hook[3].TelPos_1.TelPos := L#3;
   Front.Hook[4].HookOver := L#3805;
   Front.Hook[4].HookUnderOffset := L#115;
   Front.Hook[4].TelPos_1.TelPos := L#3;
   Front.Hook[5].HookOver := L#2835;
   Front.Hook[5].HookUnderOffset := L#115;
   Front.Hook[5].TelPos_1.TelPos := L#3;
   Front.Hook[6].HookOver := L#1865;
   Front.Hook[6].HookUnderOffset := L#115;
   Front.Hook[6].TelPos_1.TelPos := L#3;
   Rear.Hook[1].HookOver := L#6716;
   Rear.Hook[1].HookUnderOffset := L#115;
   Rear.Hook[1].TelPos_1.TelPos := L#4;
   Rear.Hook[2].HookOver := L#5745;
   Rear.Hook[2].HookUnderOffset := L#115;
   Rear.Hook[2].TelPos_1.TelPos := L#4;
   Rear.Hook[3].HookOver := L#4775;
   Rear.Hook[3].HookUnderOffset := L#115;
   Rear.Hook[3].TelPos_1.TelPos := L#4;
   Rear.Hook[4].HookOver := L#3805;
   Rear.Hook[4].HookUnderOffset := L#115;
   Rear.Hook[4].TelPos_1.TelPos := L#4;
   Rear.Hook[5].HookOver := L#2835;
   Rear.Hook[5].HookUnderOffset := L#115;
   Rear.Hook[5].TelPos_1.TelPos := L#4;
   Rear.Hook[6].HookOver := L#1865;
   Rear.Hook[6].HookUnderOffset := L#115;
   Rear.Hook[6].TelPos_1.TelPos := L#4;
END_DATA_BLOCK

DATA_BLOCK "BR03_TR03"	// DB 225
VERSION : 0.1
  STRUCT
   Front : STRUCT
    Hook : ARRAY  [1 .. 10 ] OF UDT 102;
   END_STRUCT ;
   Rear : STRUCT
    Hook : ARRAY  [1 .. 10 ] OF UDT 102;
   END_STRUCT ;
  END_STRUCT ;	
BEGIN
   Front.Hook[1].HookOver := L#6716;
   Front.Hook[1].HookUnderOffset := L#115;
   Front.Hook[1].TelPos_1.TelPos := L#3;
   Front.Hook[2].HookOver := L#5745;
   Front.Hook[2].HookUnderOffset := L#115;
   Front.Hook[2].TelPos_1.TelPos := L#3;
   Front.Hook[3].HookOver := L#4775;
   Front.Hook[3].HookUnderOffset := L#115;
   Front.Hook[3].TelPos_1.TelPos := L#3;
   Front.Hook[4].HookOver := L#3805;
   Front.Hook[4].HookUnderOffset := L#115;
   Front.Hook[4].TelPos_1.TelPos := L#3;
   Front.Hook[5].HookOver := L#2835;
   Front.Hook[5].HookUnderOffset := L#115;
   Front.Hook[5].TelPos_1.TelPos := L#3;
   Front.Hook[6].HookOver := L#1865;
   Front.Hook[6].HookUnderOffset := L#115;
   Front.Hook[6].TelPos_1.TelPos := L#3;
   Rear.Hook[1].HookOver := L#6716;
   Rear.Hook[1].HookUnderOffset := L#115;
   Rear.Hook[1].TelPos_1.TelPos := L#4;
   Rear.Hook[2].HookOver := L#5745;
   Rear.Hook[2].HookUnderOffset := L#115;
   Rear.Hook[2].TelPos_1.TelPos := L#4;
   Rear.Hook[3].HookOver := L#4775;
   Rear.Hook[3].HookUnderOffset := L#115;
   Rear.Hook[3].TelPos_1.TelPos := L#4;
   Rear.Hook[4].HookOver := L#3805;
   Rear.Hook[4].HookUnderOffset := L#115;
   Rear.Hook[4].TelPos_1.TelPos := L#4;
   Rear.Hook[5].HookOver := L#2835;
   Rear.Hook[5].HookUnderOffset := L#115;
   Rear.Hook[5].TelPos_1.TelPos := L#4;
   Rear.Hook[6].HookOver := L#1865;
   Rear.Hook[6].HookUnderOffset := L#115;
   Rear.Hook[6].TelPos_1.TelPos := L#4;
END_DATA_BLOCK

DATA_BLOCK "BR03_TR04"	// DB 226
VERSION : 0.1
  STRUCT
   Front : STRUCT
    Hook : ARRAY  [1 .. 10 ] OF UDT 102;
   END_STRUCT ;
   Rear : STRUCT
    Hook : ARRAY  [1 .. 10 ] OF UDT 102;
   END_STRUCT ;
  END_STRUCT ;	
BEGIN
   Front.Hook[1].HookOver := L#6716;
   Front.Hook[1].HookUnderOffset := L#115;
   Front.Hook[1].TelPos_1.TelPos := L#3;
   Front.Hook[2].HookOver := L#5745;
   Front.Hook[2].HookUnderOffset := L#115;
   Front.Hook[2].TelPos_1.TelPos := L#3;
   Front.Hook[3].HookOver := L#4775;
   Front.Hook[3].HookUnderOffset := L#115;
   Front.Hook[3].TelPos_1.TelPos := L#3;
   Front.Hook[4].HookOver := L#3805;
   Front.Hook[4].HookUnderOffset := L#115;
   Front.Hook[4].TelPos_1.TelPos := L#3;
   Front.Hook[5].HookOver := L#2835;
   Front.Hook[5].HookUnderOffset := L#115;
   Front.Hook[5].TelPos_1.TelPos := L#3;
   Front.Hook[6].HookOver := L#1865;
   Front.Hook[6].HookUnderOffset := L#115;
   Front.Hook[6].TelPos_1.TelPos := L#3;
   Rear.Hook[1].HookOver := L#6716;
   Rear.Hook[1].HookUnderOffset := L#115;
   Rear.Hook[1].TelPos_1.TelPos := L#4;
   Rear.Hook[2].HookOver := L#5745;
   Rear.Hook[2].HookUnderOffset := L#115;
   Rear.Hook[2].TelPos_1.TelPos := L#4;
   Rear.Hook[3].HookOver := L#4775;
   Rear.Hook[3].HookUnderOffset := L#115;
   Rear.Hook[3].TelPos_1.TelPos := L#4;
   Rear.Hook[4].HookOver := L#3805;
   Rear.Hook[4].HookUnderOffset := L#115;
   Rear.Hook[4].TelPos_1.TelPos := L#4;
   Rear.Hook[5].HookOver := L#2835;
   Rear.Hook[5].HookUnderOffset := L#115;
   Rear.Hook[5].TelPos_1.TelPos := L#4;
   Rear.Hook[6].HookOver := L#1865;
   Rear.Hook[6].HookUnderOffset := L#115;
   Rear.Hook[6].TelPos_1.TelPos := L#4;
END_DATA_BLOCK

DATA_BLOCK "BR03_TR05"	// DB 227
VERSION : 0.1
  STRUCT
   Front : STRUCT
    Hook : ARRAY  [1 .. 10 ] OF UDT 102;
   END_STRUCT ;
   Rear : STRUCT
    Hook : ARRAY  [1 .. 10 ] OF UDT 102;
   END_STRUCT ;
  END_STRUCT ;	
BEGIN
   Front.Hook[1].HookOver := L#6716;
   Front.Hook[1].HookUnderOffset := L#115;
   Front.Hook[1].TelPos_1.TelPos := L#3;
   Front.Hook[2].HookOver := L#5745;
   Front.Hook[2].HookUnderOffset := L#115;
   Front.Hook[2].TelPos_1.TelPos := L#3;
   Front.Hook[3].HookOver := L#4775;
   Front.Hook[3].HookUnderOffset := L#115;
   Front.Hook[3].TelPos_1.TelPos := L#3;
   Front.Hook[4].HookOver := L#3805;
   Front.Hook[4].HookUnderOffset := L#115;
   Front.Hook[4].TelPos_1.TelPos := L#3;
   Front.Hook[5].HookOver := L#2835;
   Front.Hook[5].HookUnderOffset := L#115;
   Front.Hook[5].TelPos_1.TelPos := L#3;
   Front.Hook[6].HookOver := L#1865;
   Front.Hook[6].HookUnderOffset := L#115;
   Front.Hook[6].TelPos_1.TelPos := L#3;
   Rear.Hook[1].HookOver := L#6716;
   Rear.Hook[1].HookUnderOffset := L#115;
   Rear.Hook[1].TelPos_1.TelPos := L#4;
   Rear.Hook[2].HookOver := L#5745;
   Rear.Hook[2].HookUnderOffset := L#115;
   Rear.Hook[2].TelPos_1.TelPos := L#4;
   Rear.Hook[3].HookOver := L#4775;
   Rear.Hook[3].HookUnderOffset := L#115;
   Rear.Hook[3].TelPos_1.TelPos := L#4;
   Rear.Hook[4].HookOver := L#3805;
   Rear.Hook[4].HookUnderOffset := L#115;
   Rear.Hook[4].TelPos_1.TelPos := L#4;
   Rear.Hook[5].HookOver := L#2835;
   Rear.Hook[5].HookUnderOffset := L#115;
   Rear.Hook[5].TelPos_1.TelPos := L#4;
   Rear.Hook[6].HookOver := L#1865;
   Rear.Hook[6].HookUnderOffset := L#115;
   Rear.Hook[6].TelPos_1.TelPos := L#4;
END_DATA_BLOCK

DATA_BLOCK "BR03_TR06"	// DB 228
VERSION : 0.1
  STRUCT
   Front : STRUCT
    Hook : ARRAY  [1 .. 10 ] OF UDT 102;
   END_STRUCT ;
   Rear : STRUCT
    Hook : ARRAY  [1 .. 10 ] OF UDT 102;
   END_STRUCT ;
  END_STRUCT ;	
BEGIN
   Front.Hook[1].HookOver := L#6716;
   Front.Hook[1].HookUnderOffset := L#115;
   Front.Hook[1].TelPos_1.TelPos := L#3;
   Front.Hook[2].HookOver := L#5745;
   Front.Hook[2].HookUnderOffset := L#115;
   Front.Hook[2].TelPos_1.TelPos := L#3;
   Front.Hook[3].HookOver := L#4775;
   Front.Hook[3].HookUnderOffset := L#115;
   Front.Hook[3].TelPos_1.TelPos := L#3;
   Front.Hook[4].HookOver := L#3805;
   Front.Hook[4].HookUnderOffset := L#115;
   Front.Hook[4].TelPos_1.TelPos := L#3;
   Front.Hook[5].HookOver := L#2835;
   Front.Hook[5].HookUnderOffset := L#115;
   Front.Hook[5].TelPos_1.TelPos := L#3;
   Front.Hook[6].HookOver := L#1865;
   Front.Hook[6].HookUnderOffset := L#115;
   Front.Hook[6].TelPos_1.TelPos := L#3;
   Rear.Hook[1].HookOver := L#6716;
   Rear.Hook[1].HookUnderOffset := L#115;
   Rear.Hook[1].TelPos_1.TelPos := L#4;
   Rear.Hook[2].HookOver := L#5745;
   Rear.Hook[2].HookUnderOffset := L#115;
   Rear.Hook[2].TelPos_1.TelPos := L#4;
   Rear.Hook[3].HookOver := L#4775;
   Rear.Hook[3].HookUnderOffset := L#115;
   Rear.Hook[3].TelPos_1.TelPos := L#4;
   Rear.Hook[4].HookOver := L#3805;
   Rear.Hook[4].HookUnderOffset := L#115;
   Rear.Hook[4].TelPos_1.TelPos := L#4;
   Rear.Hook[5].HookOver := L#2835;
   Rear.Hook[5].HookUnderOffset := L#115;
   Rear.Hook[5].TelPos_1.TelPos := L#4;
   Rear.Hook[6].HookOver := L#1865;
   Rear.Hook[6].HookUnderOffset := L#115;
   Rear.Hook[6].TelPos_1.TelPos := L#4;
END_DATA_BLOCK

DATA_BLOCK "BR03_TR07"	// DB 229
VERSION : 0.1
  STRUCT
   Front : STRUCT
    Hook : ARRAY  [1 .. 10 ] OF UDT 102;
   END_STRUCT ;
   Rear : STRUCT
    Hook : ARRAY  [1 .. 10 ] OF UDT 102;
   END_STRUCT ;
  END_STRUCT ;	
BEGIN
   Front.Hook[1].HookOver := L#6716;
   Front.Hook[1].HookUnderOffset := L#115;
   Front.Hook[1].TelPos_1.TelPos := L#3;
   Front.Hook[2].HookOver := L#5745;
   Front.Hook[2].HookUnderOffset := L#115;
   Front.Hook[2].TelPos_1.TelPos := L#3;
   Front.Hook[3].HookOver := L#4775;
   Front.Hook[3].HookUnderOffset := L#115;
   Front.Hook[3].TelPos_1.TelPos := L#3;
   Front.Hook[4].HookOver := L#3805;
   Front.Hook[4].HookUnderOffset := L#115;
   Front.Hook[4].TelPos_1.TelPos := L#3;
   Front.Hook[5].HookOver := L#2835;
   Front.Hook[5].HookUnderOffset := L#115;
   Front.Hook[5].TelPos_1.TelPos := L#3;
   Front.Hook[6].HookOver := L#1865;
   Front.Hook[6].HookUnderOffset := L#115;
   Front.Hook[6].TelPos_1.TelPos := L#3;
   Rear.Hook[1].HookOver := L#6716;
   Rear.Hook[1].HookUnderOffset := L#115;
   Rear.Hook[1].TelPos_1.TelPos := L#4;
   Rear.Hook[2].HookOver := L#5745;
   Rear.Hook[2].HookUnderOffset := L#115;
   Rear.Hook[2].TelPos_1.TelPos := L#4;
   Rear.Hook[3].HookOver := L#4775;
   Rear.Hook[3].HookUnderOffset := L#115;
   Rear.Hook[3].TelPos_1.TelPos := L#4;
   Rear.Hook[4].HookOver := L#3805;
   Rear.Hook[4].HookUnderOffset := L#115;
   Rear.Hook[4].TelPos_1.TelPos := L#4;
   Rear.Hook[5].HookOver := L#2835;
   Rear.Hook[5].HookUnderOffset := L#115;
   Rear.Hook[5].TelPos_1.TelPos := L#4;
   Rear.Hook[6].HookOver := L#1865;
   Rear.Hook[6].HookUnderOffset := L#115;
   Rear.Hook[6].TelPos_1.TelPos := L#4;
END_DATA_BLOCK

DATA_BLOCK "BR03_TR08"	// DB 230
VERSION : 0.1
  STRUCT
   Front : STRUCT
    Hook : ARRAY  [1 .. 10 ] OF UDT 102;
   END_STRUCT ;
   Rear : STRUCT
    Hook : ARRAY  [1 .. 10 ] OF UDT 102;
   END_STRUCT ;
  END_STRUCT ;	
BEGIN
   Front.Hook[1].HookOver := L#6716;
   Front.Hook[1].HookUnderOffset := L#115;
   Front.Hook[1].TelPos_1.TelPos := L#3;
   Front.Hook[2].HookOver := L#5745;
   Front.Hook[2].HookUnderOffset := L#115;
   Front.Hook[2].TelPos_1.TelPos := L#3;
   Front.Hook[3].HookOver := L#4775;
   Front.Hook[3].HookUnderOffset := L#115;
   Front.Hook[3].TelPos_1.TelPos := L#3;
   Front.Hook[4].HookOver := L#3805;
   Front.Hook[4].HookUnderOffset := L#115;
   Front.Hook[4].TelPos_1.TelPos := L#3;
   Front.Hook[5].HookOver := L#2835;
   Front.Hook[5].HookUnderOffset := L#115;
   Front.Hook[5].TelPos_1.TelPos := L#3;
   Front.Hook[6].HookOver := L#1865;
   Front.Hook[6].HookUnderOffset := L#115;
   Front.Hook[6].TelPos_1.TelPos := L#3;
   Rear.Hook[1].HookOver := L#6716;
   Rear.Hook[1].HookUnderOffset := L#115;
   Rear.Hook[1].TelPos_1.TelPos := L#4;
   Rear.Hook[2].HookOver := L#5745;
   Rear.Hook[2].HookUnderOffset := L#115;
   Rear.Hook[2].TelPos_1.TelPos := L#4;
   Rear.Hook[3].HookOver := L#4775;
   Rear.Hook[3].HookUnderOffset := L#115;
   Rear.Hook[3].TelPos_1.TelPos := L#4;
   Rear.Hook[4].HookOver := L#3805;
   Rear.Hook[4].HookUnderOffset := L#115;
   Rear.Hook[4].TelPos_1.TelPos := L#4;
   Rear.Hook[5].HookOver := L#2835;
   Rear.Hook[5].HookUnderOffset := L#115;
   Rear.Hook[5].TelPos_1.TelPos := L#4;
   Rear.Hook[6].HookOver := L#1865;
   Rear.Hook[6].HookUnderOffset := L#115;
   Rear.Hook[6].TelPos_1.TelPos := L#4;
END_DATA_BLOCK

DATA_BLOCK "BR03_TR09"	// DB 231
VERSION : 0.1
  STRUCT
   Front : STRUCT
    Hook : ARRAY  [1 .. 10 ] OF UDT 102;
   END_STRUCT ;
   Rear : STRUCT
    Hook : ARRAY  [1 .. 10 ] OF UDT 102;
   END_STRUCT ;
  END_STRUCT ;	
BEGIN
   Front.Hook[1].HookOver := L#6716;
   Front.Hook[1].HookUnderOffset := L#115;
   Front.Hook[1].TelPos_1.TelPos := L#3;
   Front.Hook[2].HookOver := L#5745;
   Front.Hook[2].HookUnderOffset := L#115;
   Front.Hook[2].TelPos_1.TelPos := L#3;
   Front.Hook[3].HookOver := L#4775;
   Front.Hook[3].HookUnderOffset := L#115;
   Front.Hook[3].TelPos_1.TelPos := L#3;
   Front.Hook[4].HookOver := L#3805;
   Front.Hook[4].HookUnderOffset := L#115;
   Front.Hook[4].TelPos_1.TelPos := L#3;
   Front.Hook[5].HookOver := L#2835;
   Front.Hook[5].HookUnderOffset := L#115;
   Front.Hook[5].TelPos_1.TelPos := L#3;
   Front.Hook[6].HookOver := L#1865;
   Front.Hook[6].HookUnderOffset := L#115;
   Front.Hook[6].TelPos_1.TelPos := L#3;
   Rear.Hook[1].HookOver := L#6716;
   Rear.Hook[1].HookUnderOffset := L#115;
   Rear.Hook[1].TelPos_1.TelPos := L#4;
   Rear.Hook[2].HookOver := L#5745;
   Rear.Hook[2].HookUnderOffset := L#115;
   Rear.Hook[2].TelPos_1.TelPos := L#4;
   Rear.Hook[3].HookOver := L#4775;
   Rear.Hook[3].HookUnderOffset := L#115;
   Rear.Hook[3].TelPos_1.TelPos := L#4;
   Rear.Hook[4].HookOver := L#3805;
   Rear.Hook[4].HookUnderOffset := L#115;
   Rear.Hook[4].TelPos_1.TelPos := L#4;
   Rear.Hook[5].HookOver := L#2835;
   Rear.Hook[5].HookUnderOffset := L#115;
   Rear.Hook[5].TelPos_1.TelPos := L#4;
   Rear.Hook[6].HookOver := L#1865;
   Rear.Hook[6].HookUnderOffset := L#115;
   Rear.Hook[6].TelPos_1.TelPos := L#4;
END_DATA_BLOCK

DATA_BLOCK "BR03_TR10"	// DB 232
VERSION : 0.1
  STRUCT
   Front : STRUCT
    Hook : ARRAY  [1 .. 10 ] OF UDT 102;
   END_STRUCT ;
   Rear : STRUCT
    Hook : ARRAY  [1 .. 10 ] OF UDT 102;
   END_STRUCT ;
  END_STRUCT ;	
BEGIN
   Front.Hook[1].HookOver := L#6716;
   Front.Hook[1].HookUnderOffset := L#115;
   Front.Hook[1].TelPos_1.TelPos := L#3;
   Front.Hook[2].HookOver := L#5745;
   Front.Hook[2].HookUnderOffset := L#115;
   Front.Hook[2].TelPos_1.TelPos := L#3;
   Front.Hook[3].HookOver := L#4775;
   Front.Hook[3].HookUnderOffset := L#115;
   Front.Hook[3].TelPos_1.TelPos := L#3;
   Front.Hook[4].HookOver := L#3805;
   Front.Hook[4].HookUnderOffset := L#115;
   Front.Hook[4].TelPos_1.TelPos := L#3;
   Front.Hook[5].HookOver := L#2835;
   Front.Hook[5].HookUnderOffset := L#115;
   Front.Hook[5].TelPos_1.TelPos := L#3;
   Rear.Hook[1].HookOver := L#6716;
   Rear.Hook[1].HookUnderOffset := L#115;
   Rear.Hook[1].TelPos_1.TelPos := L#4;
   Rear.Hook[2].HookOver := L#5745;
   Rear.Hook[2].HookUnderOffset := L#115;
   Rear.Hook[2].TelPos_1.TelPos := L#4;
   Rear.Hook[3].HookOver := L#4775;
   Rear.Hook[3].HookUnderOffset := L#115;
   Rear.Hook[3].TelPos_1.TelPos := L#4;
   Rear.Hook[4].HookOver := L#3805;
   Rear.Hook[4].HookUnderOffset := L#115;
   Rear.Hook[4].TelPos_1.TelPos := L#4;
   Rear.Hook[5].HookOver := L#2835;
   Rear.Hook[5].HookUnderOffset := L#115;
   Rear.Hook[5].TelPos_1.TelPos := L#4;
END_DATA_BLOCK

DATA_BLOCK "BR03_TR11"	// DB 233
VERSION : 0.1
  STRUCT
   Front : STRUCT
    Hook : ARRAY  [1 .. 10 ] OF UDT 102;
   END_STRUCT ;
   Rear : STRUCT
    Hook : ARRAY  [1 .. 10 ] OF UDT 102;
   END_STRUCT ;
  END_STRUCT ;	
BEGIN
   Front.Hook[1].HookOver := L#6716;
   Front.Hook[1].HookUnderOffset := L#115;
   Front.Hook[1].TelPos_1.TelPos := L#3;
   Front.Hook[2].HookOver := L#5745;
   Front.Hook[2].HookUnderOffset := L#115;
   Front.Hook[2].TelPos_1.TelPos := L#3;
   Front.Hook[3].HookOver := L#4775;
   Front.Hook[3].HookUnderOffset := L#115;
   Front.Hook[3].TelPos_1.TelPos := L#3;
   Front.Hook[4].HookOver := L#3805;
   Front.Hook[4].HookUnderOffset := L#115;
   Front.Hook[4].TelPos_1.TelPos := L#3;
   Front.Hook[5].HookOver := L#2835;
   Front.Hook[5].HookUnderOffset := L#115;
   Front.Hook[5].TelPos_1.TelPos := L#3;
   Front.Hook[6].HookOver := L#1865;
   Front.Hook[6].HookUnderOffset := L#115;
   Front.Hook[6].TelPos_1.TelPos := L#3;
   Rear.Hook[1].HookOver := L#6716;
   Rear.Hook[1].HookUnderOffset := L#115;
   Rear.Hook[1].TelPos_1.TelPos := L#4;
   Rear.Hook[2].HookOver := L#5745;
   Rear.Hook[2].HookUnderOffset := L#115;
   Rear.Hook[2].TelPos_1.TelPos := L#4;
   Rear.Hook[3].HookOver := L#4775;
   Rear.Hook[3].HookUnderOffset := L#115;
   Rear.Hook[3].TelPos_1.TelPos := L#4;
   Rear.Hook[4].HookOver := L#3805;
   Rear.Hook[4].HookUnderOffset := L#115;
   Rear.Hook[4].TelPos_1.TelPos := L#4;
   Rear.Hook[5].HookOver := L#2835;
   Rear.Hook[5].HookUnderOffset := L#115;
   Rear.Hook[5].TelPos_1.TelPos := L#4;
   Rear.Hook[6].HookOver := L#1865;
   Rear.Hook[6].HookUnderOffset := L#115;
   Rear.Hook[6].TelPos_1.TelPos := L#4;
END_DATA_BLOCK

DATA_BLOCK "BR04_TR01"	// DB 234
VERSION : 0.1
  STRUCT
   Front : STRUCT
    Hook : ARRAY  [1 .. 10 ] OF UDT 102;
   END_STRUCT ;
   Rear : STRUCT
    Hook : ARRAY  [1 .. 10 ] OF UDT 102;
   END_STRUCT ;
  END_STRUCT ;	
BEGIN
   Front.Hook[1].HookOver := L#6716;
   Front.Hook[1].HookUnderOffset := L#115;
   Front.Hook[1].TelPos_1.TelPos := L#3;
   Front.Hook[2].HookOver := L#5745;
   Front.Hook[2].HookUnderOffset := L#115;
   Front.Hook[2].TelPos_1.TelPos := L#3;
   Front.Hook[3].HookOver := L#4775;
   Front.Hook[3].HookUnderOffset := L#115;
   Front.Hook[3].TelPos_1.TelPos := L#3;
   Front.Hook[4].HookOver := L#3805;
   Front.Hook[4].HookUnderOffset := L#115;
   Front.Hook[4].TelPos_1.TelPos := L#3;
   Front.Hook[5].HookOver := L#2835;
   Front.Hook[5].HookUnderOffset := L#115;
   Front.Hook[5].TelPos_1.TelPos := L#3;
   Rear.Hook[1].HookOver := L#6716;
   Rear.Hook[1].HookUnderOffset := L#115;
   Rear.Hook[1].TelPos_1.TelPos := L#4;
   Rear.Hook[2].HookOver := L#5745;
   Rear.Hook[2].HookUnderOffset := L#115;
   Rear.Hook[2].TelPos_1.TelPos := L#4;
   Rear.Hook[3].HookOver := L#4775;
   Rear.Hook[3].HookUnderOffset := L#115;
   Rear.Hook[3].TelPos_1.TelPos := L#4;
   Rear.Hook[4].HookOver := L#3805;
   Rear.Hook[4].HookUnderOffset := L#115;
   Rear.Hook[4].TelPos_1.TelPos := L#4;
   Rear.Hook[5].HookOver := L#2835;
   Rear.Hook[5].HookUnderOffset := L#115;
   Rear.Hook[5].TelPos_1.TelPos := L#4;
END_DATA_BLOCK

DATA_BLOCK "BR04_TR02"	// DB 235
VERSION : 0.1
  STRUCT
   Front : STRUCT
    Hook : ARRAY  [1 .. 10 ] OF UDT 102;
   END_STRUCT ;
   Rear : STRUCT
    Hook : ARRAY  [1 .. 10 ] OF UDT 102;
   END_STRUCT ;
  END_STRUCT ;	
BEGIN
   Front.Hook[1].HookOver := L#6716;
   Front.Hook[1].HookUnderOffset := L#115;
   Front.Hook[1].TelPos_1.TelPos := L#3;
   Front.Hook[2].HookOver := L#5745;
   Front.Hook[2].HookUnderOffset := L#115;
   Front.Hook[2].TelPos_1.TelPos := L#3;
   Front.Hook[3].HookOver := L#4775;
   Front.Hook[3].HookUnderOffset := L#115;
   Front.Hook[3].TelPos_1.TelPos := L#3;
   Front.Hook[4].HookOver := L#3805;
   Front.Hook[4].HookUnderOffset := L#115;
   Front.Hook[4].TelPos_1.TelPos := L#3;
   Front.Hook[5].HookOver := L#2835;
   Front.Hook[5].HookUnderOffset := L#115;
   Front.Hook[5].TelPos_1.TelPos := L#3;
   Front.Hook[6].HookOver := L#1865;
   Front.Hook[6].HookUnderOffset := L#115;
   Front.Hook[6].TelPos_1.TelPos := L#3;
   Rear.Hook[1].HookOver := L#6716;
   Rear.Hook[1].HookUnderOffset := L#115;
   Rear.Hook[1].TelPos_1.TelPos := L#4;
   Rear.Hook[2].HookOver := L#5745;
   Rear.Hook[2].HookUnderOffset := L#115;
   Rear.Hook[2].TelPos_1.TelPos := L#4;
   Rear.Hook[3].HookOver := L#4775;
   Rear.Hook[3].HookUnderOffset := L#115;
   Rear.Hook[3].TelPos_1.TelPos := L#4;
   Rear.Hook[4].HookOver := L#3805;
   Rear.Hook[4].HookUnderOffset := L#115;
   Rear.Hook[4].TelPos_1.TelPos := L#4;
   Rear.Hook[5].HookOver := L#2835;
   Rear.Hook[5].HookUnderOffset := L#115;
   Rear.Hook[5].TelPos_1.TelPos := L#4;
   Rear.Hook[6].HookOver := L#1865;
   Rear.Hook[6].HookUnderOffset := L#115;
   Rear.Hook[6].TelPos_1.TelPos := L#4;
END_DATA_BLOCK

DATA_BLOCK "BR04_TR03"	// DB 236
VERSION : 0.1
  STRUCT
   Front : STRUCT
    Hook : ARRAY  [1 .. 10 ] OF UDT 102;
   END_STRUCT ;
   Rear : STRUCT
    Hook : ARRAY  [1 .. 10 ] OF UDT 102;
   END_STRUCT ;
  END_STRUCT ;	
BEGIN
   Front.Hook[1].HookOver := L#6716;
   Front.Hook[1].HookUnderOffset := L#115;
   Front.Hook[1].TelPos_1.TelPos := L#3;
   Front.Hook[2].HookOver := L#5745;
   Front.Hook[2].HookUnderOffset := L#115;
   Front.Hook[2].TelPos_1.TelPos := L#3;
   Front.Hook[3].HookOver := L#4775;
   Front.Hook[3].HookUnderOffset := L#115;
   Front.Hook[3].TelPos_1.TelPos := L#3;
   Front.Hook[4].HookOver := L#3805;
   Front.Hook[4].HookUnderOffset := L#115;
   Front.Hook[4].TelPos_1.TelPos := L#3;
   Front.Hook[5].HookOver := L#2835;
   Front.Hook[5].HookUnderOffset := L#115;
   Front.Hook[5].TelPos_1.TelPos := L#3;
   Front.Hook[6].HookOver := L#1865;
   Front.Hook[6].HookUnderOffset := L#115;
   Front.Hook[6].TelPos_1.TelPos := L#3;
   Rear.Hook[1].HookOver := L#6716;
   Rear.Hook[1].HookUnderOffset := L#115;
   Rear.Hook[1].TelPos_1.TelPos := L#4;
   Rear.Hook[2].HookOver := L#5745;
   Rear.Hook[2].HookUnderOffset := L#115;
   Rear.Hook[2].TelPos_1.TelPos := L#4;
   Rear.Hook[3].HookOver := L#4775;
   Rear.Hook[3].HookUnderOffset := L#115;
   Rear.Hook[3].TelPos_1.TelPos := L#4;
   Rear.Hook[4].HookOver := L#3805;
   Rear.Hook[4].HookUnderOffset := L#115;
   Rear.Hook[4].TelPos_1.TelPos := L#4;
   Rear.Hook[5].HookOver := L#2835;
   Rear.Hook[5].HookUnderOffset := L#115;
   Rear.Hook[5].TelPos_1.TelPos := L#4;
   Rear.Hook[6].HookOver := L#1865;
   Rear.Hook[6].HookUnderOffset := L#115;
   Rear.Hook[6].TelPos_1.TelPos := L#4;
END_DATA_BLOCK

DATA_BLOCK "BR04_TR04"	// DB 237
VERSION : 0.1
  STRUCT
   Front : STRUCT
    Hook : ARRAY  [1 .. 10 ] OF UDT 102;
   END_STRUCT ;
   Rear : STRUCT
    Hook : ARRAY  [1 .. 10 ] OF UDT 102;
   END_STRUCT ;
  END_STRUCT ;	
BEGIN
   Front.Hook[1].HookOver := L#6716;
   Front.Hook[1].HookUnderOffset := L#115;
   Front.Hook[1].TelPos_1.TelPos := L#3;
   Front.Hook[2].HookOver := L#5745;
   Front.Hook[2].HookUnderOffset := L#115;
   Front.Hook[2].TelPos_1.TelPos := L#3;
   Front.Hook[3].HookOver := L#4775;
   Front.Hook[3].HookUnderOffset := L#115;
   Front.Hook[3].TelPos_1.TelPos := L#3;
   Front.Hook[4].HookOver := L#3805;
   Front.Hook[4].HookUnderOffset := L#115;
   Front.Hook[4].TelPos_1.TelPos := L#3;
   Front.Hook[5].HookOver := L#2835;
   Front.Hook[5].HookUnderOffset := L#115;
   Front.Hook[5].TelPos_1.TelPos := L#3;
   Front.Hook[6].HookOver := L#1865;
   Front.Hook[6].HookUnderOffset := L#115;
   Front.Hook[6].TelPos_1.TelPos := L#3;
   Rear.Hook[1].HookOver := L#6716;
   Rear.Hook[1].HookUnderOffset := L#115;
   Rear.Hook[1].TelPos_1.TelPos := L#4;
   Rear.Hook[2].HookOver := L#5745;
   Rear.Hook[2].HookUnderOffset := L#115;
   Rear.Hook[2].TelPos_1.TelPos := L#4;
   Rear.Hook[3].HookOver := L#4775;
   Rear.Hook[3].HookUnderOffset := L#115;
   Rear.Hook[3].TelPos_1.TelPos := L#4;
   Rear.Hook[4].HookOver := L#3805;
   Rear.Hook[4].HookUnderOffset := L#115;
   Rear.Hook[4].TelPos_1.TelPos := L#4;
   Rear.Hook[5].HookOver := L#2835;
   Rear.Hook[5].HookUnderOffset := L#115;
   Rear.Hook[5].TelPos_1.TelPos := L#4;
   Rear.Hook[6].HookOver := L#1865;
   Rear.Hook[6].HookUnderOffset := L#115;
   Rear.Hook[6].TelPos_1.TelPos := L#4;
END_DATA_BLOCK

DATA_BLOCK "BR04_TR05"	// DB 238
VERSION : 0.1
  STRUCT
   Front : STRUCT
    Hook : ARRAY  [1 .. 10 ] OF UDT 102;
   END_STRUCT ;
   Rear : STRUCT
    Hook : ARRAY  [1 .. 10 ] OF UDT 102;
   END_STRUCT ;
  END_STRUCT ;	
BEGIN
   Front.Hook[1].HookOver := L#6716;
   Front.Hook[1].HookUnderOffset := L#115;
   Front.Hook[1].TelPos_1.TelPos := L#3;
   Front.Hook[2].HookOver := L#5745;
   Front.Hook[2].HookUnderOffset := L#115;
   Front.Hook[2].TelPos_1.TelPos := L#3;
   Front.Hook[3].HookOver := L#4775;
   Front.Hook[3].HookUnderOffset := L#115;
   Front.Hook[3].TelPos_1.TelPos := L#3;
   Front.Hook[4].HookOver := L#3805;
   Front.Hook[4].HookUnderOffset := L#115;
   Front.Hook[4].TelPos_1.TelPos := L#3;
   Front.Hook[5].HookOver := L#2835;
   Front.Hook[5].HookUnderOffset := L#115;
   Front.Hook[5].TelPos_1.TelPos := L#3;
   Front.Hook[6].HookOver := L#1865;
   Front.Hook[6].HookUnderOffset := L#115;
   Front.Hook[6].TelPos_1.TelPos := L#3;
   Rear.Hook[1].HookOver := L#6716;
   Rear.Hook[1].HookUnderOffset := L#115;
   Rear.Hook[1].TelPos_1.TelPos := L#4;
   Rear.Hook[2].HookOver := L#5745;
   Rear.Hook[2].HookUnderOffset := L#115;
   Rear.Hook[2].TelPos_1.TelPos := L#4;
   Rear.Hook[3].HookOver := L#4775;
   Rear.Hook[3].HookUnderOffset := L#115;
   Rear.Hook[3].TelPos_1.TelPos := L#4;
   Rear.Hook[4].HookOver := L#3805;
   Rear.Hook[4].HookUnderOffset := L#115;
   Rear.Hook[4].TelPos_1.TelPos := L#4;
   Rear.Hook[5].HookOver := L#2835;
   Rear.Hook[5].HookUnderOffset := L#115;
   Rear.Hook[5].TelPos_1.TelPos := L#4;
   Rear.Hook[6].HookOver := L#1865;
   Rear.Hook[6].HookUnderOffset := L#115;
   Rear.Hook[6].TelPos_1.TelPos := L#4;
END_DATA_BLOCK

DATA_BLOCK "BR04_TR06"	// DB 239
VERSION : 0.1
  STRUCT
   Front : STRUCT
    Hook : ARRAY  [1 .. 10 ] OF UDT 102;
   END_STRUCT ;
   Rear : STRUCT
    Hook : ARRAY  [1 .. 10 ] OF UDT 102;
   END_STRUCT ;
  END_STRUCT ;	
BEGIN
   Front.Hook[1].HookOver := L#6716;
   Front.Hook[1].HookUnderOffset := L#115;
   Front.Hook[1].TelPos_1.TelPos := L#3;
   Front.Hook[2].HookOver := L#5745;
   Front.Hook[2].HookUnderOffset := L#115;
   Front.Hook[2].TelPos_1.TelPos := L#3;
   Front.Hook[3].HookOver := L#4775;
   Front.Hook[3].HookUnderOffset := L#115;
   Front.Hook[3].TelPos_1.TelPos := L#3;
   Front.Hook[4].HookOver := L#3805;
   Front.Hook[4].HookUnderOffset := L#115;
   Front.Hook[4].TelPos_1.TelPos := L#3;
   Front.Hook[5].HookOver := L#2835;
   Front.Hook[5].HookUnderOffset := L#115;
   Front.Hook[5].TelPos_1.TelPos := L#3;
   Front.Hook[6].HookOver := L#1865;
   Front.Hook[6].HookUnderOffset := L#115;
   Front.Hook[6].TelPos_1.TelPos := L#3;
   Rear.Hook[1].HookOver := L#6716;
   Rear.Hook[1].HookUnderOffset := L#115;
   Rear.Hook[1].TelPos_1.TelPos := L#4;
   Rear.Hook[2].HookOver := L#5745;
   Rear.Hook[2].HookUnderOffset := L#115;
   Rear.Hook[2].TelPos_1.TelPos := L#4;
   Rear.Hook[3].HookOver := L#4775;
   Rear.Hook[3].HookUnderOffset := L#115;
   Rear.Hook[3].TelPos_1.TelPos := L#4;
   Rear.Hook[4].HookOver := L#3805;
   Rear.Hook[4].HookUnderOffset := L#115;
   Rear.Hook[4].TelPos_1.TelPos := L#4;
   Rear.Hook[5].HookOver := L#2835;
   Rear.Hook[5].HookUnderOffset := L#115;
   Rear.Hook[5].TelPos_1.TelPos := L#4;
   Rear.Hook[6].HookOver := L#1865;
   Rear.Hook[6].HookUnderOffset := L#115;
   Rear.Hook[6].TelPos_1.TelPos := L#4;
END_DATA_BLOCK

